C03638=1064.079,67.653,428.198,172.244,27.907,155.137
C03639=1064.085,67.903,428.181,172.246,27.909,155.137
C03640=1064.091,68.152,428.163,172.246,27.912,155.138
C03641=1064.097,68.401,428.146,172.248,27.915,155.138
C03642=1064.103,68.650,428.128,172.249,27.917,155.139
C03643=1064.109,68.899,428.111,172.251,27.920,155.139
C03644=1064.115,69.150,428.094,172.252,27.923,155.139
C03645=1064.120,69.399,428.076,172.254,27.925,155.140
C03646=1064.127,69.648,428.059,172.256,27.928,155.140
C03647=1064.133,69.897,428.041,172.257,27.931,155.141
C03648=1064.138,70.146,428.024,172.259,27.934,155.141
C03649=1064.144,70.396,428.006,172.259,27.936,155.141
C03650=1064.150,70.645,427.989,172.261,27.939,155.142
C03651=1064.157,70.894,427.971,172.262,27.941,155.142
C03652=1064.162,71.143,427.953,172.264,27.944,155.142
C03653=1064.168,71.393,427.935,172.265,27.947,155.143
C03654=1064.174,71.642,427.918,172.267,27.950,155.143
C03655=1064.180,71.891,427.901,172.269,27.952,155.144
C03656=1064.186,72.141,427.883,172.270,27.955,155.144
C03657=1064.192,72.390,427.865,172.272,27.958,155.144
C03658=1064.198,72.640,427.847,172.272,27.961,155.145
C03659=1064.203,72.889,427.830,172.274,27.963,155.145
C03660=1064.210,73.138,427.812,172.275,27.966,155.146
C03661=1064.216,73.387,427.795,172.277,27.968,155.146
C03662=1064.222,73.637,427.777,172.279,27.971,155.146
C03663=1064.227,73.886,427.759,172.280,27.974,155.147
C03664=1064.233,74.136,427.741,172.282,27.977,155.147
C03665=1064.239,74.385,427.724,172.283,27.980,155.147
C03666=1064.245,74.634,427.706,172.285,27.982,155.148
C03667=1064.251,74.883,427.689,172.285,27.984,155.148
C03668=1064.257,75.133,427.671,172.287,27.987,155.149
C03669=1064.263,75.382,427.653,172.289,27.990,155.149
C03670=1064.269,75.632,427.636,172.290,27.993,155.149
C03671=1064.275,75.881,427.618,172.292,27.996,155.150
C03672=1064.281,76.130,427.599,172.293,27.998,155.150
C03673=1064.287,76.379,427.582,172.295,28.001,155.151
C03674=1064.293,76.629,427.564,172.296,28.003,155.151
C03675=1064.299,76.877,427.547,172.298,28.006,155.151
C03676=1064.305,77.127,427.529,172.299,28.009,155.152
C03677=1064.311,77.376,427.511,172.300,28.011,155.152
C03678=1064.317,77.626,427.493,172.302,28.014,155.152
C03679=1064.323,77.874,427.475,172.303,28.017,155.153
C03680=1064.329,78.159,427.455,172.305,28.020,155.153
C03681=1064.336,78.442,427.434,172.307,28.023,155.154
C03682=1064.343,78.726,427.414,172.309,28.026,155.154
C03683=1064.349,79.010,427.394,172.310,28.029,155.155
C03684=1064.355,79.259,427.376,172.312,28.032,155.155
C03685=1064.361,79.508,427.358,172.313,28.035,155.155
C03686=1064.367,79.757,427.340,172.315,28.037,155.156
C03687=1064.373,80.007,427.322,172.315,28.040,155.156
C03688=1064.379,80.256,427.304,172.317,28.043,155.157
C03689=1064.384,80.506,427.286,172.319,28.046,155.157
C03690=1064.390,80.755,427.267,172.320,28.048,155.157
C03691=1064.396,81.004,427.249,172.322,28.051,155.158
C03692=1064.402,81.254,427.232,172.323,28.054,155.158
C03693=1064.408,81.503,427.213,172.325,28.057,155.159
C03694=1064.414,81.752,427.196,172.326,28.059,155.159
C03695=1064.420,82.001,427.178,172.328,28.062,155.159
C03696=1064.426,82.250,427.159,172.329,28.065,155.160
C03697=1064.432,82.500,427.142,172.330,28.068,155.160
C03698=1064.437,82.750,427.123,172.332,28.070,155.161
C03699=1064.443,82.998,427.105,172.333,28.073,155.161
C03700=1064.449,83.248,427.087,172.335,28.075,155.161
C03701=1064.455,83.497,427.069,172.336,28.078,155.162
C03702=1064.461,83.746,427.051,172.338,28.081,155.162
C03703=1064.467,83.996,427.033,172.339,28.084,155.162
C03704=1064.473,84.245,427.015,172.341,28.087,155.163
C03705=1064.479,84.494,426.996,172.343,28.089,155.163
C03706=1064.484,84.743,426.978,172.344,28.092,155.164
C03707=1064.490,84.992,426.960,172.346,28.095,155.164
C03708=1064.497,85.242,426.942,172.346,28.097,155.165
C03709=1064.502,85.491,426.924,172.348,28.100,155.165
C03710=1064.509,85.740,426.905,172.350,28.102,155.165
C03711=1064.515,85.990,426.888,172.351,28.105,155.166
C03712=1064.520,86.239,426.869,172.353,28.108,155.166
C03713=1064.526,86.488,426.851,172.354,28.111,155.166
C03714=1064.532,86.738,426.832,172.356,28.114,155.167
C03715=1064.538,86.987,426.814,172.357,28.116,155.167
C03716=1064.544,87.236,426.796,172.359,28.119,155.168
C03717=1064.550,87.485,426.778,172.360,28.122,155.168
C03718=1064.555,87.734,426.759,172.362,28.124,155.168
C03719=1064.562,87.984,426.741,172.364,28.127,155.169
C03720=1064.568,88.233,426.722,172.364,28.129,155.169
C03721=1064.574,88.482,426.705,172.366,28.132,155.170
C03722=1064.580,88.731,426.686,172.367,28.135,155.170
C03723=1064.585,88.981,426.668,172.369,28.138,155.170
C03724=1064.591,89.230,426.649,172.370,28.141,155.171
C03725=1064.597,89.479,426.631,172.372,28.143,155.171
C03726=1064.604,89.729,426.613,172.374,28.146,155.171
C03727=1064.610,89.978,426.594,172.375,28.148,155.172
C03728=1064.615,90.227,426.576,172.377,28.151,155.172
C03729=1064.621,90.476,426.557,172.378,28.154,155.173
C03730=1064.627,90.726,426.539,172.380,28.157,155.173
C03731=1064.633,90.974,426.521,172.382,28.159,155.173
C03732=1064.639,91.224,426.502,172.382,28.162,155.174
C03733=1064.645,91.474,426.484,172.384,28.165,155.174
C03734=1064.650,91.722,426.465,172.385,28.168,155.175
C03735=1064.657,91.971,426.446,172.387,28.170,155.175
C03736=1064.663,92.221,426.429,172.388,28.173,155.175
C03737=1064.668,92.471,426.409,172.390,28.175,155.176
C03738=1064.674,92.719,426.391,172.392,28.178,155.176
C03739=1064.680,92.969,426.372,172.393,28.181,155.177
C03740=1064.686,93.218,426.354,172.395,28.184,155.177
C03741=1064.691,93.467,426.335,172.396,28.186,155.177
C03742=1064.697,93.717,426.317,172.398,28.189,155.178
C03743=1064.704,93.966,426.298,172.399,28.192,155.178
C03744=1064.710,94.250,426.277,172.401,28.195,155.179
C03745=1064.716,94.533,426.256,172.402,28.198,155.179
C03746=1064.724,94.817,426.234,172.404,28.201,155.180
C03747=1064.730,95.101,426.213,172.406,28.204,155.180
C03748=1064.736,95.351,426.195,172.407,28.207,155.180
C03749=1064.742,95.599,426.177,172.409,28.210,155.181
C03750=1064.747,95.848,426.157,172.410,28.213,155.181
C03751=1064.754,96.098,426.139,172.412,28.215,155.182
C03752=1064.760,96.347,426.119,172.413,28.218,155.182
C03753=1064.765,96.596,426.102,172.415,28.221,155.182
C03754=1064.771,96.845,426.083,172.416,28.224,155.183
C03755=1064.777,97.095,426.064,172.418,28.226,155.183
C03756=1064.783,97.344,426.045,172.420,28.229,155.183
C03757=1064.789,97.593,426.026,172.421,28.231,155.184
C03758=1064.794,97.842,426.007,172.423,28.234,155.184
C03759=1064.801,98.092,425.989,172.424,28.237,155.185
C03760=1064.806,98.341,425.970,172.426,28.240,155.185
C03761=1064.813,98.590,425.951,172.428,28.243,155.185
C03762=1064.818,98.840,425.932,172.429,28.245,155.186
C03763=1064.824,99.088,425.914,172.430,28.248,155.186
C03764=1064.830,99.337,425.895,172.431,28.251,155.187
C03765=1064.836,99.587,425.876,172.433,28.253,155.187
C03766=1064.842,99.836,425.857,172.435,28.256,155.187
C03767=1064.848,100.085,425.838,172.436,28.258,155.188
C03768=1064.854,100.335,425.819,172.438,28.261,155.188
C03769=1064.860,100.584,425.801,172.439,28.264,155.189
C03770=1064.865,100.833,425.782,172.441,28.267,155.189
C03771=1064.872,101.082,425.763,172.442,28.269,155.189
C03772=1064.877,101.332,425.744,172.444,28.272,155.190
C03773=1064.884,101.581,425.725,172.446,28.275,155.190
C03774=1064.889,101.830,425.706,172.447,28.278,155.191
C03775=1064.895,102.079,425.687,172.449,28.281,155.191
C03776=1064.900,102.328,425.668,172.450,28.283,155.191
C03777=1064.907,102.577,425.649,172.452,28.286,155.192
C03778=1064.912,102.827,425.630,172.453,28.289,155.192
C03779=1064.918,103.076,425.611,172.455,28.292,155.193
C03780=1064.924,103.325,425.592,172.457,28.294,155.193
C03781=1064.930,103.574,425.573,172.458,28.297,155.193
C03782=1064.936,103.823,425.553,172.460,28.300,155.194
C03783=1064.941,104.072,425.534,172.460,28.302,155.194
C03784=1064.948,104.322,425.516,172.462,28.305,155.195
C03785=1064.953,104.571,425.496,172.464,28.307,155.195
C03786=1064.959,104.820,425.477,172.465,28.310,155.195
C03787=1064.965,105.070,425.458,172.467,28.313,155.196
C03788=1064.971,105.318,425.440,172.468,28.316,155.196
C03789=1064.976,105.568,425.420,172.470,28.318,155.197
C03790=1064.982,105.817,425.401,172.471,28.321,155.197
C03791=1064.988,106.066,425.381,172.473,28.324,155.197
C03792=1064.994,106.315,425.362,172.475,28.327,155.198
C03793=1065.000,106.564,425.343,172.476,28.330,155.198
C03794=1065.006,106.814,425.324,172.478,28.332,155.199
C03795=1065.011,107.063,425.305,172.479,28.335,155.199
C03796=1065.018,107.312,425.286,172.481,28.338,155.199
C03797=1065.024,107.561,425.266,172.483,28.341,155.200
C03798=1065.030,107.811,425.247,172.484,28.343,155.200
C03799=1065.035,108.059,425.228,172.486,28.346,155.201
C03800=1065.041,108.309,425.209,172.487,28.349,155.201
C03801=1065.047,108.558,425.190,172.489,28.352,155.201
C03802=1065.053,108.807,425.170,172.491,28.354,155.202
C03803=1065.058,109.056,425.151,172.492,28.357,155.202
C03804=1065.064,109.306,425.132,172.494,28.359,155.202
C03805=1065.071,109.555,425.113,172.495,28.362,155.203
C03806=1065.077,109.804,425.093,172.497,28.365,155.203
C03807=1065.082,110.053,425.074,172.498,28.368,155.204
C03808=1065.089,110.337,425.052,172.500,28.370,155.204
C03809=1065.096,110.621,425.030,172.502,28.374,155.205
C03810=1065.102,110.904,425.008,172.503,28.377,155.205
C03811=1065.109,111.189,424.985,172.506,28.380,155.205
C03812=1065.115,111.438,424.966,172.507,28.383,155.206
C03813=1065.121,111.688,424.947,172.509,28.386,155.206
C03814=1065.128,111.936,424.928,172.510,28.388,155.207
C03815=1065.133,112.185,424.908,172.512,28.391,155.207
C03816=1065.138,112.434,424.889,172.513,28.394,155.207
C03817=1065.144,112.683,424.870,172.515,28.397,155.208
C03818=1065.150,112.932,424.850,172.517,28.399,155.208
C03819=1065.156,113.181,424.830,172.518,28.402,155.209
C03820=1065.162,113.431,424.811,172.520,28.404,155.209
C03821=1065.167,113.680,424.792,172.521,28.407,155.209
C03822=1065.173,113.929,424.772,172.523,28.410,155.210
C03823=1065.179,114.178,424.753,172.525,28.413,155.210
C03824=1065.185,114.427,424.733,172.526,28.415,155.211
C03825=1065.191,114.677,424.713,172.528,28.418,155.211
C03826=1065.197,114.925,424.693,172.529,28.421,155.211
C03827=1065.202,115.175,424.674,172.531,28.424,155.212
C03828=1065.208,115.424,424.654,172.533,28.426,155.212
C03829=1065.213,115.673,424.634,172.534,28.430,155.213
C03830=1065.219,115.923,424.615,172.536,28.433,155.213
C03831=1065.225,116.172,424.595,172.537,28.435,155.214
C03832=1065.231,116.420,424.575,172.539,28.438,155.214
C03833=1065.237,116.670,424.556,172.540,28.441,155.214
C03834=1065.242,116.919,424.535,172.542,28.444,155.215
C03835=1065.248,117.168,424.516,172.544,28.446,155.215
C03836=1065.254,117.417,424.496,172.545,28.449,155.216
C03837=1065.259,117.667,424.477,172.547,28.452,155.216
C03838=1065.265,117.916,424.457,172.548,28.455,155.216
C03839=1065.271,118.165,424.438,172.550,28.457,155.217
C03840=1065.276,118.414,424.417,172.552,28.460,155.217
C03841=1065.282,118.663,424.397,172.553,28.463,155.218
C03842=1065.288,118.912,424.378,172.555,28.466,155.218
C03843=1065.294,119.161,424.358,172.556,28.468,155.218
C03844=1065.300,119.411,424.339,172.558,28.471,155.219
C03845=1065.306,119.660,424.318,172.560,28.474,155.219
C03846=1065.312,119.909,424.298,172.561,28.477,155.220
C03847=1065.317,120.159,424.279,172.563,28.479,155.220
C03848=1065.323,120.407,424.259,172.564,28.482,155.220
C03849=1065.329,120.656,424.239,172.566,28.485,155.221
C03850=1065.334,120.906,424.219,172.568,28.488,155.221
C03851=1065.340,121.155,424.199,172.569,28.490,155.222
C03852=1065.346,121.404,424.179,172.571,28.493,155.222
C03853=1065.352,121.653,424.160,172.572,28.496,155.222
C03854=1065.358,121.902,424.140,172.574,28.499,155.223
C03855=1065.363,122.151,424.119,172.575,28.501,155.223
C03856=1065.369,122.401,424.100,172.577,28.504,155.224
C03857=1065.375,122.650,424.080,172.579,28.507,155.224
C03858=1065.381,122.899,424.060,172.580,28.510,155.224
C03859=1065.387,123.148,424.039,172.582,28.512,155.225
C03860=1065.392,123.397,424.020,172.583,28.515,155.225
C03861=1065.398,123.646,424.000,172.585,28.518,155.226
C03862=1065.404,123.895,423.980,172.587,28.521,155.226
C03863=1065.410,124.144,423.960,172.588,28.523,155.226
C03864=1065.416,124.394,423.940,172.590,28.526,155.227
C03865=1065.422,124.643,423.920,172.591,28.529,155.227
C03866=1065.428,124.892,423.900,172.593,28.532,155.228
C03867=1065.434,125.141,423.880,172.595,28.534,155.228
C03868=1065.439,125.390,423.859,172.596,28.537,155.228
C03869=1065.445,125.639,423.840,172.598,28.539,155.229
C03870=1065.451,125.889,423.820,172.600,28.542,155.229
C03871=1065.457,126.138,423.800,172.601,28.545,155.230
C03872=1065.463,126.421,423.776,172.604,28.548,155.230
C03873=1065.470,126.705,423.754,172.605,28.551,155.230
C03874=1065.477,126.989,423.731,172.607,28.554,155.231
C03875=1065.484,127.272,423.708,172.609,28.557,155.231
C03876=1065.489,127.521,423.688,172.611,28.560,155.232
C03877=1065.496,127.771,423.667,172.612,28.563,155.232
C03878=1065.502,128.019,423.647,172.614,28.566,155.233
C03879=1065.507,128.269,423.628,172.616,28.568,155.233
C03880=1065.513,128.518,423.608,172.617,28.571,155.233
C03881=1065.519,128.767,423.587,172.619,28.574,155.234
C03882=1065.525,129.016,423.567,172.620,28.577,155.234
C03883=1065.531,129.265,423.547,172.622,28.579,155.235
C03884=1065.537,129.514,423.527,172.624,28.582,155.235
C03885=1065.543,129.764,423.507,172.625,28.584,155.235
C03886=1065.548,130.013,423.486,172.627,28.587,155.236
C03887=1065.554,130.262,423.466,172.629,28.590,155.236
C03888=1065.560,130.510,423.446,172.630,28.593,155.237
C03889=1065.566,130.760,423.425,172.632,28.595,155.237
C03890=1065.572,131.009,423.405,172.634,28.598,155.237
C03891=1065.578,131.258,423.385,172.636,28.601,155.238
C03892=1065.584,131.508,423.364,172.638,28.604,155.238
C03893=1065.590,131.757,423.344,172.639,28.607,155.239
C03894=1065.596,132.005,423.324,172.641,28.609,155.239
C03895=1065.601,132.254,423.304,172.642,28.612,155.239
C03896=1065.608,132.504,423.283,172.644,28.615,155.240
C03897=1065.614,132.753,423.262,172.646,28.617,155.240
C03898=1065.619,133.002,423.242,172.647,28.620,155.241
C03899=1065.625,133.250,423.222,172.649,28.623,155.241
C03900=1065.631,133.500,423.201,172.650,28.626,155.241
C03901=1065.637,133.749,423.181,172.652,28.628,155.242
C03902=1065.642,133.998,423.160,172.654,28.631,155.242
C03903=1065.648,134.247,423.140,172.656,28.634,155.243
C03904=1065.654,134.496,423.119,172.658,28.637,155.243
C03905=1065.659,134.745,423.098,172.659,28.640,155.243
C03906=1065.665,134.994,423.078,172.661,28.642,155.244
C03907=1065.671,135.244,423.057,172.663,28.645,155.244
C03908=1065.677,135.493,423.037,172.664,28.648,155.245
C03909=1065.682,135.742,423.017,172.666,28.651,155.245
C03910=1065.689,135.991,422.996,172.667,28.653,155.245
C03911=1065.695,136.240,422.975,172.669,28.656,155.246
C03912=1065.700,136.489,422.955,172.671,28.659,155.246
C03913=1065.706,136.739,422.934,172.672,28.662,155.247
C03914=1065.712,136.987,422.913,172.675,28.665,155.247
C03915=1065.718,137.236,422.893,172.676,28.667,155.247
C03916=1065.724,137.486,422.872,172.678,28.670,155.248
C03917=1065.729,137.735,422.852,172.680,28.673,155.248
C03918=1065.735,137.983,422.831,172.681,28.675,155.249
C03919=1065.741,138.233,422.810,172.683,28.678,155.249
C03920=1065.747,138.482,422.789,172.684,28.681,155.249
C03921=1065.753,138.730,422.769,172.686,28.684,155.250
C03922=1065.759,138.980,422.748,172.688,28.686,155.250
C03923=1065.764,139.229,422.727,172.689,28.689,155.251
C03924=1065.770,139.477,422.707,172.692,28.692,155.251
C03925=1065.776,139.727,422.686,172.693,28.695,155.251
C03926=1065.781,139.976,422.665,172.695,28.698,155.252
C03927=1065.788,140.224,422.644,172.697,28.700,155.252
C03928=1065.793,140.474,422.624,172.698,28.703,155.253
C03929=1065.799,140.723,422.603,172.700,28.706,155.253
C03930=1065.805,140.973,422.581,172.702,28.709,155.253
C03931=1065.810,141.222,422.561,172.703,28.711,155.254
C03932=1065.816,141.470,422.540,172.705,28.714,155.254
C03933=1065.822,141.720,422.519,172.707,28.717,155.255
C03934=1065.828,141.968,422.498,172.709,28.720,155.255
C03935=1065.833,142.217,422.477,172.711,28.722,155.255
C03936=1065.840,142.501,422.453,172.712,28.726,155.256
C03937=1065.846,142.785,422.430,172.715,28.729,155.256
C03938=1065.853,143.069,422.406,172.716,28.732,155.257
C03939=1065.860,143.351,422.382,172.718,28.735,155.257
C03940=1065.866,143.601,422.361,172.720,28.738,155.258
C03941=1065.871,143.850,422.340,172.722,28.741,155.258
C03942=1065.877,144.099,422.319,172.724,28.744,155.259
C03943=1065.883,144.348,422.298,172.725,28.746,155.259
C03944=1065.889,144.598,422.277,172.727,28.749,155.259
C03945=1065.894,144.846,422.255,172.728,28.752,155.260
C03946=1065.900,145.095,422.235,172.730,28.755,155.260
C03947=1065.906,145.344,422.214,172.733,28.758,155.261
C03948=1065.912,145.593,422.193,172.734,28.760,155.261
C03949=1065.918,145.843,422.172,172.736,28.763,155.261
C03950=1065.923,146.091,422.150,172.737,28.766,155.262
C03951=1065.929,146.341,422.129,172.739,28.769,155.262
C03952=1065.935,146.589,422.108,172.741,28.771,155.263
C03953=1065.941,146.839,422.088,172.742,28.774,155.263
C03954=1065.947,147.087,422.067,172.745,28.777,155.263
C03955=1065.953,147.337,422.045,172.746,28.780,155.264
C03956=1065.958,147.586,422.024,172.748,28.782,155.264
C03957=1065.964,147.835,422.003,172.750,28.785,155.265
C03958=1065.970,148.083,421.981,172.751,28.788,155.265
C03959=1065.976,148.333,421.961,172.753,28.791,155.265
C03960=1065.981,148.582,421.939,172.756,28.794,155.266
C03961=1065.988,148.831,421.918,172.757,28.796,155.266
C03962=1065.993,149.080,421.897,172.759,28.799,155.267
C03963=1065.999,149.329,421.875,172.760,28.802,155.267
C03964=1066.005,149.578,421.854,172.762,28.804,155.267
C03965=1066.011,149.827,421.833,172.764,28.807,155.268
C03966=1066.016,150.076,421.812,172.766,28.810,155.268
C03967=1066.022,150.325,421.790,172.768,28.813,155.269
C03968=1066.028,150.574,421.769,172.769,28.816,155.269
C03969=1066.034,150.823,421.747,172.771,28.819,155.270
C03970=1066.039,151.072,421.726,172.773,28.822,155.270
C03971=1066.045,151.321,421.705,172.774,28.824,155.270
C03972=1066.050,151.570,421.683,172.777,28.827,155.271
C03973=1066.056,151.819,421.662,172.778,28.830,155.271
C03974=1066.062,152.068,421.640,172.780,28.833,155.272
C03975=1066.068,152.317,421.619,172.782,28.835,155.272
C03976=1066.074,152.566,421.598,172.783,28.838,155.272
C03977=1066.079,152.815,421.577,172.786,28.841,155.273
C03978=1066.085,153.064,421.555,172.788,28.844,155.273
C03979=1066.091,153.313,421.534,172.789,28.847,155.274
C03980=1066.097,153.562,421.512,172.791,28.850,155.274
C03981=1066.102,153.811,421.490,172.792,28.853,155.275
C03982=1066.108,154.060,421.469,172.794,28.855,155.275
C03983=1066.114,154.309,421.447,172.797,28.858,155.275
C03984=1066.120,154.558,421.426,172.798,28.861,155.276
C03985=1066.126,154.807,421.404,172.800,28.864,155.276
C03986=1066.132,155.056,421.383,172.801,28.866,155.277
C03987=1066.138,155.306,421.362,172.803,28.869,155.277
C03988=1066.142,155.554,421.340,172.806,28.872,155.277
C03989=1066.149,155.804,421.318,172.807,28.875,155.278
C03990=1066.154,156.052,421.297,172.809,28.878,155.278
C03991=1066.160,156.301,421.275,172.811,28.880,155.279
C03992=1066.166,156.551,421.253,172.813,28.884,155.279
C03993=1066.171,156.799,421.232,172.815,28.887,155.280
C03994=1066.177,157.049,421.210,172.816,28.889,155.280
C03995=1066.183,157.297,421.189,172.818,28.892,155.280
C03996=1066.189,157.546,421.166,172.820,28.895,155.281
C03997=1066.195,157.795,421.145,172.822,28.898,155.281
C03998=1066.200,158.044,421.123,172.824,28.900,155.282
C03999=1066.206,158.293,421.101,172.825,28.903,155.282
C04000=1066.213,158.577,421.076,172.828,28.907,155.282
C04001=1066.219,158.859,421.052,172.830,28.910,155.283
C04002=1066.226,159.143,421.027,172.832,28.913,155.283
C04003=1066.233,159.427,421.002,172.834,28.916,155.284
C04004=1066.238,159.675,420.981,172.835,28.919,155.284
C04005=1066.244,159.924,420.959,172.838,28.922,155.285
C04006=1066.250,160.174,420.937,172.840,28.924,155.285
C04007=1066.255,160.422,420.916,172.841,28.927,155.286
C04008=1066.261,160.671,420.894,172.843,28.930,155.286
C04009=1066.267,160.921,420.872,172.845,28.933,155.286
C04010=1066.273,161.169,420.850,172.847,28.936,155.287
C04011=1066.279,161.418,420.828,172.849,28.939,155.287
C04012=1066.284,161.668,420.806,172.850,28.942,155.288
C04013=1066.289,161.916,420.784,172.853,28.944,155.288
C04014=1066.296,162.165,420.762,172.854,28.948,155.289
C04015=1066.300,162.414,420.740,172.856,28.950,155.289
C04016=1066.307,162.663,420.718,172.858,28.953,155.289
C04017=1066.312,162.913,420.696,172.859,28.956,155.290
C04018=1066.317,163.161,420.673,172.862,28.959,155.290
C04019=1066.323,163.410,420.652,172.863,28.962,155.291
C04020=1066.329,163.659,420.629,172.865,28.965,155.291
C04021=1066.334,163.908,420.607,172.867,28.968,155.292
C04022=1066.340,164.157,420.585,172.869,28.971,155.292
C04023=1066.345,164.406,420.563,172.871,28.974,155.292
C04024=1066.351,164.655,420.540,172.873,28.976,155.293
C04025=1066.357,164.904,420.519,172.874,28.980,155.293
C04026=1066.362,165.153,420.497,172.877,28.983,155.294
C04027=1066.368,165.401,420.475,172.878,28.985,155.294
C04028=1066.374,165.651,420.452,172.880,28.988,155.295
C04029=1066.379,165.900,420.430,172.883,28.992,155.295
C04030=1066.385,166.148,420.408,172.884,28.994,155.295
C04031=1066.390,166.398,420.386,172.886,28.997,155.296
C04032=1066.396,166.647,420.363,172.887,29.000,155.296
C04033=1066.402,166.895,420.342,172.890,29.003,155.297
C04034=1066.407,167.144,420.319,172.892,29.006,155.297
C04035=1066.413,167.393,420.296,172.893,29.009,155.298
C04036=1066.419,167.642,420.274,172.895,29.011,155.298
C04037=1066.424,167.891,420.252,172.897,29.015,155.299
C04038=1066.429,168.140,420.230,172.899,29.018,155.299
C04039=1066.435,168.389,420.207,172.901,29.020,155.299
C04040=1066.441,168.638,420.185,172.903,29.023,155.300
C04041=1066.446,168.887,420.163,172.905,29.026,155.300
C04042=1066.452,169.136,420.140,172.907,29.029,155.301
C04043=1066.458,169.385,420.118,172.908,29.032,155.301
C04044=1066.464,169.634,420.095,172.911,29.035,155.301
C04045=1066.469,169.882,420.073,172.912,29.038,155.302
C04046=1066.475,170.131,420.051,172.914,29.041,155.302
C04047=1066.481,170.381,420.029,172.917,29.044,155.303
C04048=1066.487,170.629,420.006,172.918,29.046,155.303
C04049=1066.492,170.879,419.984,172.920,29.049,155.304
C04050=1066.498,171.127,419.962,172.922,29.053,155.304
C04051=1066.504,171.376,419.939,172.924,29.055,155.305
C04052=1066.509,171.625,419.917,172.926,29.058,155.305
C04053=1066.515,171.874,419.894,172.927,29.061,155.305
C04054=1066.521,172.123,419.871,172.930,29.064,155.306
C04055=1066.527,172.372,419.849,172.932,29.067,155.306
C04056=1066.532,172.620,419.826,172.933,29.070,155.307
C04057=1066.538,172.869,419.804,172.936,29.073,155.307
C04058=1066.544,173.119,419.782,172.937,29.075,155.307
C04059=1066.549,173.367,419.759,172.939,29.079,155.308
C04060=1066.555,173.616,419.736,172.942,29.081,155.308
C04061=1066.561,173.866,419.714,172.943,29.084,155.309
C04062=1066.567,174.114,419.691,172.945,29.087,155.309
C04063=1066.573,174.363,419.668,172.947,29.090,155.310
C04064=1066.579,174.646,419.643,172.949,29.093,155.310
C04065=1066.586,174.929,419.618,172.952,29.097,155.311
C04066=1066.592,175.212,419.592,172.954,29.100,155.311
C04067=1066.598,175.495,419.566,172.956,29.103,155.312
C04068=1066.604,175.744,419.543,172.958,29.106,155.312
C04069=1066.610,175.992,419.521,172.960,29.109,155.312
C04070=1066.616,176.241,419.498,172.962,29.112,155.313
C04071=1066.622,176.491,419.476,172.964,29.115,155.313
C04072=1066.627,176.739,419.453,172.966,29.118,155.314
C04073=1066.633,176.988,419.430,172.968,29.121,155.314
C04074=1066.640,177.237,419.408,172.970,29.123,155.315
C04075=1066.645,177.486,419.385,172.972,29.126,155.315
C04076=1066.651,177.735,419.362,172.974,29.130,155.316
C04077=1066.657,177.984,419.339,172.976,29.132,155.316
C04078=1066.662,178.233,419.317,172.978,29.135,155.316
C04079=1066.669,178.482,419.294,172.980,29.138,155.317
C04080=1066.674,178.731,419.271,172.982,29.141,155.317
C04081=1066.680,178.980,419.248,172.983,29.144,155.318
C04082=1066.686,179.228,419.225,172.986,29.147,155.318
C04083=1066.692,179.477,419.202,172.988,29.149,155.318
C04084=1066.697,179.726,419.180,172.990,29.152,155.319
C04085=1066.704,179.975,419.157,172.992,29.155,155.319
C04086=1066.710,180.224,419.134,172.994,29.158,155.320
C04087=1066.715,180.473,419.111,172.996,29.161,155.320
C04088=1066.721,180.722,419.088,172.998,29.164,155.321
C04089=1066.727,180.970,419.065,173.000,29.167,155.321
C04090=1066.732,181.219,419.042,173.002,29.170,155.321
C04091=1066.739,181.468,419.020,173.004,29.173,155.322
C04092=1066.745,181.717,418.997,173.006,29.176,155.322
C04093=1066.750,181.966,418.974,173.008,29.178,155.323
C04094=1066.756,182.215,418.951,173.011,29.181,155.323
C04095=1066.762,182.464,418.928,173.012,29.184,155.324
C04096=1066.768,182.713,418.905,173.014,29.187,155.324
C04097=1066.775,182.962,418.883,173.016,29.190,155.324
C04098=1066.780,183.211,418.860,173.018,29.193,155.325
C04099=1066.786,183.459,418.837,173.021,29.196,155.325
C04100=1066.792,183.708,418.814,173.022,29.198,155.326
C04101=1066.798,183.957,418.790,173.025,29.201,155.326
C04102=1066.804,184.206,418.767,173.027,29.205,155.327
C04103=1066.809,184.454,418.744,173.028,29.207,155.327
C04104=1066.816,184.704,418.721,173.031,29.210,155.327
C04105=1066.821,184.953,418.698,173.032,29.213,155.328
C04106=1066.827,185.202,418.675,173.035,29.216,155.328
C04107=1066.832,185.450,418.651,173.037,29.219,155.329
C04108=1066.838,185.699,418.628,173.038,29.222,155.329
C04109=1066.844,185.948,418.605,173.041,29.225,155.330
C04110=1066.849,186.197,418.581,173.043,29.228,155.330
C04111=1066.855,186.446,418.558,173.045,29.231,155.331
C04112=1066.861,186.695,418.535,173.047,29.235,155.331
C04113=1066.866,186.944,418.511,173.049,29.238,155.331
C04114=1066.871,187.193,418.488,173.051,29.241,155.332
C04115=1066.877,187.441,418.465,173.053,29.243,155.332
C04116=1066.883,187.690,418.442,173.055,29.247,155.333
C04117=1066.888,187.939,418.418,173.057,29.250,155.333
C04118=1066.894,188.187,418.394,173.059,29.253,155.334
C04119=1066.899,188.437,418.371,173.061,29.256,155.334
C04120=1066.905,188.685,418.348,173.064,29.259,155.335
C04121=1066.911,188.934,418.324,173.065,29.262,155.335
C04122=1066.916,189.183,418.301,173.068,29.265,155.336
C04123=1066.922,189.431,418.277,173.070,29.268,155.336
C04124=1066.928,189.681,418.254,173.071,29.271,155.337
C04125=1066.933,189.930,418.230,173.074,29.274,155.337
C04126=1066.939,190.178,418.207,173.075,29.277,155.337
C04127=1066.945,190.427,418.184,173.078,29.280,155.338
C04128=1066.951,190.710,418.156,173.081,29.284,155.338
C04129=1066.958,190.992,418.130,173.082,29.287,155.339
C04130=1066.964,191.274,418.103,173.085,29.291,155.340
C04131=1066.971,191.557,418.076,173.087,29.294,155.340
C04132=1066.976,191.806,418.053,173.089,29.297,155.341
C04133=1066.982,192.055,418.029,173.092,29.300,155.341
C04134=1066.987,192.303,418.006,173.093,29.303,155.341
C04135=1066.994,192.552,417.982,173.096,29.306,155.342
C04136=1066.999,192.802,417.958,173.097,29.310,155.342
C04137=1067.005,193.050,417.934,173.100,29.312,155.343
C04138=1067.011,193.299,417.912,173.102,29.315,155.343
C04139=1067.016,193.547,417.887,173.104,29.319,155.344
C04140=1067.022,193.797,417.864,173.106,29.321,155.344
C04141=1067.028,194.046,417.840,173.108,29.325,155.345
C04142=1067.034,194.294,417.816,173.110,29.327,155.345
C04143=1067.039,194.543,417.792,173.113,29.331,155.346
C04144=1067.045,194.791,417.769,173.114,29.334,155.346
C04145=1067.051,195.041,417.746,173.117,29.337,155.346
C04146=1067.056,195.290,417.721,173.119,29.340,155.347
C04147=1067.062,195.538,417.698,173.121,29.343,155.347
C04148=1067.067,195.787,417.674,173.123,29.346,155.348
C04149=1067.074,196.036,417.650,173.125,29.349,155.348
C04150=1067.079,196.285,417.626,173.127,29.352,155.349
C04151=1067.085,196.533,417.602,173.130,29.355,155.349
C04152=1067.092,196.782,417.579,173.131,29.358,155.350
C04153=1067.097,197.031,417.555,173.134,29.362,155.350
C04154=1067.103,197.279,417.531,173.136,29.364,155.351
C04155=1067.108,197.529,417.507,173.138,29.368,155.351
C04156=1067.115,197.778,417.483,173.141,29.371,155.352
C04157=1067.120,198.026,417.459,173.142,29.373,155.352
C04158=1067.126,198.274,417.435,173.145,29.377,155.352
C04159=1067.132,198.524,417.411,173.147,29.379,155.353
C04160=1067.138,198.773,417.388,173.149,29.383,155.353
C04161=1067.143,199.021,417.364,173.151,29.386,155.354
C04162=1067.150,199.270,417.340,173.154,29.389,155.354
C04163=1067.155,199.519,417.315,173.155,29.392,155.355
C04164=1067.161,199.767,417.292,173.158,29.395,155.355
C04165=1067.166,200.017,417.268,173.160,29.398,155.356
C04166=1067.173,200.265,417.244,173.162,29.401,155.356
C04167=1067.178,200.514,417.219,173.165,29.404,155.357
C04168=1067.184,200.763,417.196,173.166,29.407,155.357
C04169=1067.190,201.011,417.172,173.169,29.410,155.357
C04170=1067.196,201.260,417.147,173.171,29.413,155.358
C04171=1067.202,201.509,417.123,173.173,29.416,155.358
C04172=1067.208,201.758,417.099,173.175,29.420,155.359
C04173=1067.214,202.006,417.075,173.177,29.422,155.359
C04174=1067.220,202.255,417.051,173.180,29.426,155.360
C04175=1067.226,202.504,417.027,173.182,29.429,155.360
C04176=1067.231,202.753,417.002,173.184,29.432,155.361
C04177=1067.237,203.001,416.979,173.186,29.435,155.361
C04178=1067.243,203.250,416.954,173.189,29.438,155.362
C04179=1067.248,203.499,416.930,173.190,29.441,155.362
C04180=1067.253,203.747,416.906,173.193,29.445,155.363
C04181=1067.259,203.997,416.881,173.195,29.448,155.363
C04182=1067.265,204.245,416.857,173.197,29.451,155.364
C04183=1067.271,204.494,416.833,173.200,29.454,155.364
C04184=1067.277,204.743,416.808,173.201,29.457,155.365
C04185=1067.282,204.991,416.784,173.204,29.460,155.365
C04186=1067.288,205.240,416.760,173.206,29.464,155.366
C04187=1067.294,205.489,416.736,173.208,29.467,155.366
C04188=1067.300,205.738,416.711,173.211,29.470,155.367
C04189=1067.305,205.987,416.687,173.212,29.473,155.367
C04190=1067.311,206.235,416.662,173.215,29.477,155.368
C04191=1067.317,206.484,416.638,173.218,29.480,155.368
C04192=1067.341,207.529,416.535,173.367,29.555,155.372
C04193=1067.347,207.746,416.513,173.369,29.559,155.373
C04194=1067.352,207.964,416.491,173.370,29.562,155.373
C04195=1067.357,208.181,416.469,173.372,29.566,155.374
C04196=1067.362,208.398,416.447,173.374,29.569,155.375
C04197=1067.367,208.615,416.425,173.375,29.573,155.375
C04198=1067.372,208.833,416.403,173.377,29.576,155.376
C04199=1067.377,209.050,416.381,173.379,29.580,155.376
C04200=1067.382,209.268,416.359,173.381,29.583,155.377
C04201=1067.389,209.516,416.333,173.383,29.587,155.378
C04202=1067.394,209.764,416.308,173.385,29.592,155.379
C04203=1067.400,210.013,416.283,173.387,29.596,155.379
C04204=1067.407,210.262,416.258,173.389,29.600,155.380
C04205=1067.413,210.511,416.233,173.391,29.604,155.381
C04206=1067.418,210.760,416.207,173.392,29.608,155.381
C04207=1067.424,211.009,416.182,173.395,29.612,155.382
C04208=1067.430,211.257,416.157,173.396,29.616,155.383
C04209=1067.436,211.505,416.131,173.399,29.620,155.383
C04210=1067.442,211.754,416.106,173.400,29.624,155.384
C04211=1067.448,212.003,416.080,173.403,29.628,155.385
C04212=1067.454,212.252,416.055,173.405,29.632,155.385
C04213=1067.460,212.500,416.030,173.407,29.636,155.386
C04214=1067.466,212.749,416.004,173.409,29.640,155.387
C04215=1067.471,212.997,415.979,173.411,29.644,155.387
C04216=1067.477,213.246,415.953,173.413,29.648,155.388
C04217=1067.484,213.495,415.928,173.415,29.652,155.389
C04218=1067.489,213.744,415.902,173.417,29.657,155.390
C04219=1067.496,213.992,415.876,173.419,29.661,155.390
C04220=1067.501,214.241,415.850,173.421,29.665,155.391
C04221=1067.507,214.489,415.825,173.423,29.669,155.392
C04222=1067.513,214.737,415.800,173.425,29.673,155.392
C04223=1067.518,214.986,415.774,173.427,29.677,155.393
C04224=1067.525,215.235,415.748,173.429,29.681,155.394
C04225=1067.530,215.484,415.723,173.431,29.685,155.395
C04226=1067.537,215.732,415.696,173.433,29.689,155.395
C04227=1067.543,215.981,415.671,173.435,29.693,155.396
C04228=1067.548,216.230,415.645,173.437,29.697,155.397
C04229=1067.554,216.478,415.620,173.439,29.701,155.397
C04230=1067.560,216.727,415.594,173.441,29.705,155.398
C04231=1067.566,216.975,415.568,173.443,29.709,155.399
C04232=1067.573,217.224,415.543,173.446,29.714,155.399
C04233=1067.578,217.473,415.517,173.447,29.717,155.400
C04234=1067.584,217.721,415.492,173.450,29.721,155.401
C04235=1067.589,217.969,415.465,173.451,29.726,155.401
C04236=1067.596,218.218,415.440,173.454,29.730,155.402
C04237=1067.601,218.467,415.414,173.455,29.733,155.403
C04238=1067.608,218.715,415.388,173.458,29.738,155.404
C04239=1067.613,218.964,415.362,173.459,29.742,155.404
C04240=1067.619,219.213,415.336,173.462,29.746,155.405
C04241=1067.625,219.461,415.310,173.465,29.749,155.405
C04242=1067.631,219.710,415.284,173.466,29.754,155.406
C04243=1067.637,219.958,415.259,173.469,29.758,155.407
C04244=1067.643,220.207,415.232,173.470,29.762,155.408
C04245=1067.649,220.455,415.207,173.473,29.766,155.408
C04246=1067.656,220.705,415.181,173.474,29.770,155.409
C04247=1067.662,220.953,415.155,173.477,29.774,155.410
C04248=1067.667,221.202,415.129,173.479,29.777,155.410
C04249=1067.673,221.421,415.105,173.480,29.781,155.411
C04250=1067.678,221.640,415.083,173.483,29.785,155.411
C04251=1067.683,221.860,415.060,173.484,29.788,155.412
C04252=1067.688,222.080,415.037,173.486,29.792,155.413
C04253=1067.693,222.299,415.013,173.488,29.795,155.413
C04254=1067.699,222.519,414.991,173.490,29.799,155.414
C04255=1067.704,222.739,414.968,173.492,29.802,155.415
C04256=1067.709,222.959,414.944,173.494,29.806,155.415
C04257=1067.715,223.207,414.918,173.496,29.810,155.416
C04258=1067.721,223.456,414.892,173.498,29.814,155.417
C04259=1067.726,223.705,414.866,173.500,29.818,155.417
C04260=1067.733,223.953,414.840,173.502,29.822,155.418
C04261=1067.738,224.202,414.814,173.504,29.827,155.419
C04262=1067.744,224.450,414.787,173.506,29.830,155.419
C04263=1067.751,224.698,414.761,173.509,29.834,155.420
C04264=1067.756,224.947,414.735,173.511,29.839,155.421
C04265=1067.762,225.195,414.709,173.513,29.843,155.421
C04266=1067.768,225.444,414.682,173.515,29.846,155.422
C04267=1067.774,225.692,414.657,173.517,29.850,155.423
C04268=1067.780,225.941,414.630,173.519,29.855,155.424
C04269=1067.786,226.190,414.603,173.521,29.858,155.424
C04270=1067.792,226.439,414.577,173.524,29.862,155.425
C04271=1067.798,226.687,414.551,173.526,29.866,155.425
C04272=1067.804,226.935,414.524,173.528,29.871,155.426
C04273=1067.809,227.184,414.498,173.530,29.875,155.427
C04274=1067.815,227.433,414.472,173.532,29.878,155.428
C04275=1067.822,227.681,414.445,173.534,29.882,155.428
C04276=1067.828,227.930,414.419,173.536,29.887,155.429
C04277=1067.833,228.179,414.393,173.539,29.891,155.430
C04278=1067.839,228.427,414.366,173.541,29.894,155.430
C04279=1067.846,228.675,414.340,173.543,29.898,155.431
C04280=1067.852,228.923,414.313,173.545,29.903,155.432
C04281=1067.858,229.172,414.286,173.547,29.906,155.432
C04282=1067.863,229.421,414.260,173.550,29.910,155.433
C04283=1067.869,229.670,414.234,173.552,29.914,155.434
C04284=1067.876,229.918,414.208,173.554,29.918,155.434
C04285=1067.882,230.167,414.181,173.556,29.922,155.435
C04286=1067.888,230.415,414.154,173.558,29.926,155.436
C04287=1067.894,230.664,414.127,173.560,29.930,155.436
C04288=1067.899,230.912,414.101,173.563,29.935,155.437
C04289=1067.905,231.160,414.074,173.565,29.938,155.438
C04290=1067.912,231.409,414.047,173.567,29.942,155.438
C04291=1067.917,231.658,414.020,173.569,29.946,155.439
C04292=1067.923,231.906,413.994,173.571,29.951,155.440
C04293=1067.929,232.154,413.967,173.574,29.954,155.441
C04294=1067.935,232.403,413.940,173.576,29.958,155.441
C04295=1067.941,232.652,413.913,173.578,29.962,155.442
C04296=1067.947,232.900,413.887,173.580,29.966,155.443
C04297=1067.953,233.149,413.860,173.582,29.970,155.443
C04298=1067.958,233.397,413.833,173.585,29.974,155.444
C04299=1067.965,233.646,413.806,173.587,29.978,155.445
C04300=1067.970,233.894,413.780,173.589,29.982,155.445
C04301=1067.976,234.143,413.753,173.592,29.986,155.446
C04302=1067.981,234.391,413.726,173.593,29.990,155.447
C04303=1067.988,234.640,413.699,173.596,29.995,155.447
C04304=1067.993,234.889,413.672,173.598,29.998,155.448
C04305=1067.999,235.104,413.649,173.600,30.002,155.449
C04306=1068.004,235.320,413.626,173.602,30.005,155.449
C04307=1068.009,235.535,413.603,173.604,30.009,155.450
C04308=1068.014,235.751,413.579,173.606,30.013,155.450
C04309=1068.019,235.966,413.555,173.608,30.016,155.451
C04310=1068.024,236.181,413.532,173.609,30.019,155.452
C04311=1068.029,236.397,413.508,173.612,30.023,155.452
C04312=1068.035,236.613,413.485,173.614,30.026,155.453
C04313=1068.041,236.861,413.458,173.615,30.030,155.454
C04314=1068.046,237.110,413.431,173.618,30.034,155.454
C04315=1068.052,237.358,413.404,173.621,30.038,155.455
C04316=1068.058,237.607,413.377,173.622,30.042,155.456
C04317=1068.064,237.855,413.350,173.625,30.046,155.456
C04318=1068.071,238.104,413.323,173.627,30.050,155.457
C04319=1068.077,238.352,413.296,173.629,30.054,155.458
C04320=1068.082,238.600,413.269,173.632,30.058,155.458
C04321=1068.088,238.850,413.241,173.634,30.062,155.459
C04322=1068.094,239.098,413.214,173.636,30.066,155.460
C04323=1068.100,239.346,413.187,173.638,30.070,155.460
C04324=1068.106,239.595,413.160,173.641,30.074,155.461
C04325=1068.112,239.843,413.133,173.643,30.078,155.462
C04326=1068.118,240.092,413.105,173.645,30.081,155.462
C04327=1068.124,240.340,413.078,173.648,30.086,155.463
C04328=1068.130,240.588,413.051,173.649,30.090,155.464
C04329=1068.136,240.837,413.024,173.652,30.094,155.464
C04330=1068.142,241.085,412.996,173.655,30.097,155.465
C04331=1068.148,241.334,412.969,173.657,30.101,155.466
C04332=1068.154,241.582,412.942,173.659,30.106,155.466
C04333=1068.160,241.831,412.915,173.661,30.110,155.467
C04334=1068.166,242.079,412.887,173.664,30.113,155.468
C04335=1068.172,242.328,412.860,173.666,30.117,155.468
C04336=1068.178,242.576,412.833,173.668,30.121,155.469
C04337=1068.183,242.825,412.805,173.671,30.126,155.470
C04338=1068.190,243.073,412.778,173.673,30.129,155.470
C04339=1068.195,243.322,412.750,173.675,30.133,155.471
C04340=1068.202,243.570,412.723,173.678,30.138,155.472
C04341=1068.207,243.818,412.695,173.680,30.142,155.473
C04342=1068.213,244.067,412.668,173.682,30.145,155.473
C04343=1068.220,244.315,412.640,173.685,30.149,155.474
C04344=1068.225,244.564,412.613,173.687,30.154,155.475
C04345=1068.231,244.812,412.585,173.689,30.157,155.475
C04346=1068.237,245.060,412.557,173.691,30.161,155.476
C04347=1068.243,245.309,412.530,173.694,30.165,155.477
C04348=1068.248,245.557,412.502,173.697,30.170,155.477
C04349=1068.255,245.806,412.475,173.698,30.173,155.478
C04350=1068.260,246.054,412.447,173.701,30.177,155.479
C04351=1068.267,246.303,412.420,173.704,30.181,155.479
C04352=1068.272,246.551,412.392,173.705,30.185,155.480
C04353=1068.279,246.799,412.364,173.708,30.189,155.481
C04354=1068.284,247.047,412.336,173.710,30.193,155.481
C04355=1068.290,247.297,412.308,173.713,30.197,155.482
C04356=1068.296,247.545,412.281,173.715,30.201,155.483
C04357=1068.302,247.793,412.253,173.717,30.205,155.483
C04358=1068.307,248.041,412.225,173.720,30.210,155.484
C04359=1068.314,248.290,412.197,173.723,30.214,155.485
C04360=1068.319,248.538,412.169,173.724,30.217,155.486
C04361=1068.324,248.751,412.145,173.727,30.221,155.486
C04362=1068.329,248.963,412.122,173.729,30.224,155.487
C04363=1068.334,249.175,412.097,173.730,30.227,155.487
C04364=1068.339,249.388,412.074,173.733,30.231,155.488
C04365=1068.344,249.601,412.050,173.735,30.235,155.489
C04366=1068.349,249.812,412.026,173.736,30.238,155.489
C04367=1068.354,250.025,412.002,173.739,30.242,155.490
C04368=1068.358,250.237,411.978,173.741,30.245,155.490
C04369=1068.365,250.486,411.951,173.743,30.249,155.491
C04370=1068.370,250.734,411.923,173.746,30.253,155.492
C04371=1068.376,250.983,411.894,173.747,30.257,155.492
C04372=1068.382,251.231,411.867,173.750,30.261,155.493
C04373=1068.388,251.479,411.839,173.753,30.265,155.494
C04374=1068.394,251.728,411.810,173.755,30.269,155.494
C04375=1068.400,251.976,411.783,173.757,30.273,155.495
C04376=1068.406,252.224,411.753,173.760,30.277,155.496
C04377=1068.412,252.472,411.726,173.762,30.281,155.497
C04378=1068.418,252.721,411.698,173.765,30.285,155.497
C04379=1068.424,252.969,411.669,173.767,30.289,155.498
C04380=1068.429,253.217,411.641,173.769,30.293,155.499
C04381=1068.436,253.466,411.614,173.772,30.297,155.499
C04382=1068.442,253.715,411.585,173.774,30.301,155.500
C04383=1068.447,253.963,411.557,173.777,30.305,155.501
C04384=1068.453,254.211,411.529,173.779,30.309,155.501
C04385=1068.459,254.459,411.500,173.781,30.313,155.502
C04386=1068.465,254.707,411.473,173.784,30.317,155.503
C04387=1068.471,254.956,411.444,173.787,30.321,155.503
C04388=1068.477,255.205,411.416,173.789,30.325,155.504
C04389=1068.483,255.453,411.388,173.791,30.329,155.505
C04390=1068.489,255.701,411.359,173.793,30.333,155.505
C04391=1068.496,255.949,411.331,173.796,30.336,155.506
C04392=1068.501,256.197,411.303,173.799,30.341,155.507
C04393=1068.507,256.446,411.275,173.801,30.345,155.508
C04394=1068.513,256.694,411.246,173.803,30.348,155.508
C04395=1068.519,256.943,411.218,173.806,30.352,155.509
C04396=1068.525,257.191,411.190,173.808,30.356,155.509
C04397=1068.531,257.439,411.161,173.811,30.361,155.510
C04398=1068.537,257.688,411.133,173.814,30.365,155.511
C04399=1068.543,257.936,411.105,173.816,30.368,155.512
C04400=1068.549,258.184,411.076,173.818,30.372,155.512
C04401=1068.555,258.433,411.048,173.821,30.376,155.513
C04402=1068.561,258.681,411.019,173.823,30.380,155.514
C04403=1068.568,258.929,410.991,173.826,30.384,155.514
C04404=1068.574,259.178,410.963,173.828,30.388,155.515
C04405=1068.579,259.425,410.934,173.831,30.392,155.516
C04406=1068.585,259.674,410.906,173.833,30.396,155.516
C04407=1068.592,259.922,410.877,173.835,30.400,155.517
C04408=1068.597,260.171,410.848,173.838,30.404,155.518
C04409=1068.604,260.419,410.819,173.841,30.408,155.518
C04410=1068.610,260.668,410.791,173.843,30.412,155.519
C04411=1068.616,260.915,410.763,173.846,30.416,155.520
C04412=1068.622,261.164,410.734,173.849,30.419,155.520
C04413=1068.628,261.412,410.705,173.850,30.424,155.521
C04414=1068.634,261.661,410.677,173.853,30.428,155.522
C04415=1068.640,261.909,410.648,173.856,30.431,155.522
C04416=1068.646,262.157,410.620,173.858,30.435,155.523
C04417=1068.652,262.368,410.595,173.860,30.438,155.524
C04418=1068.657,262.579,410.572,173.863,30.442,155.524
C04419=1068.662,262.791,410.546,173.864,30.445,155.525
C04420=1068.667,263.002,410.523,173.867,30.449,155.525
C04421=1068.673,263.213,410.498,173.869,30.452,155.526
C04422=1068.678,263.424,410.473,173.872,30.455,155.526
C04423=1068.683,263.636,410.449,173.873,30.459,155.527
C04424=1068.688,263.847,410.424,173.876,30.462,155.528
C04425=1068.694,264.095,410.396,173.878,30.466,155.528
C04426=1068.700,264.343,410.367,173.880,30.470,155.529
C04427=1068.706,264.591,410.338,173.883,30.474,155.530
C04428=1068.712,264.839,410.309,173.886,30.478,155.530
C04429=1068.717,265.088,410.280,173.888,30.482,155.531
C04430=1068.724,265.336,410.251,173.891,30.486,155.532
C04431=1068.730,265.584,410.222,173.894,30.490,155.533
C04432=1068.736,265.833,410.193,173.896,30.495,155.533
C04433=1068.742,266.081,410.163,173.899,30.498,155.534
C04434=1068.748,266.330,410.135,173.901,30.502,155.535
C04435=1068.753,266.577,410.106,173.903,30.506,155.535
C04436=1068.759,266.825,410.077,173.906,30.510,155.536
C04437=1068.765,267.074,410.047,173.909,30.514,155.537
C04438=1068.771,267.322,410.018,173.911,30.518,155.537
C04439=1068.777,267.570,409.989,173.914,30.522,155.538
C04440=1068.784,267.818,409.960,173.916,30.526,155.539
C04441=1068.789,268.067,409.931,173.919,30.530,155.539
C04442=1068.795,268.315,409.902,173.922,30.535,155.540
C04443=1068.802,268.563,409.873,173.924,30.538,155.541
C04444=1068.808,268.811,409.844,173.927,30.542,155.542
C04445=1068.813,269.059,409.814,173.929,30.546,155.542
C04446=1068.820,269.308,409.785,173.931,30.550,155.543
C04447=1068.826,269.556,409.756,173.934,30.554,155.544
C04448=1068.831,269.804,409.726,173.937,30.558,155.544
C04449=1068.838,270.052,409.697,173.939,30.562,155.545
C04450=1068.844,270.300,409.668,173.942,30.566,155.546
C04451=1068.849,270.549,409.639,173.945,30.570,155.546
C04452=1068.856,270.797,409.609,173.947,30.575,155.547
C04453=1068.861,271.045,409.580,173.950,30.578,155.548
C04454=1068.867,271.294,409.551,173.953,30.582,155.549
C04455=1068.874,271.542,409.522,173.955,30.587,155.549
C04456=1068.879,271.790,409.492,173.958,30.590,155.550
C04457=1068.886,272.038,409.462,173.961,30.594,155.551
C04458=1068.891,272.286,409.433,173.963,30.599,155.551
C04459=1068.898,272.534,409.404,173.966,30.603,155.552
C04460=1068.903,272.783,409.374,173.968,30.606,155.553
C04461=1068.909,273.031,409.345,173.970,30.611,155.553
C04462=1068.915,273.279,409.315,173.973,30.614,155.554
C04463=1068.921,273.527,409.286,173.976,30.619,155.555
C04464=1068.927,273.775,409.256,173.978,30.623,155.556
C04465=1068.933,274.023,409.227,173.981,30.627,155.556
C04466=1068.939,274.271,409.197,173.984,30.631,155.557
C04467=1068.945,274.519,409.168,173.986,30.635,155.558
C04468=1068.951,274.768,409.138,173.989,30.639,155.558
C04469=1068.958,275.016,409.108,173.992,30.643,155.559
C04470=1068.963,275.264,409.078,173.994,30.647,155.560
C04471=1068.969,275.513,409.049,173.997,30.651,155.561
C04472=1068.975,275.760,409.019,174.000,30.655,155.561
C04473=1068.980,275.973,408.993,174.003,30.659,155.562
C04474=1068.986,276.186,408.968,174.004,30.662,155.562
C04475=1068.991,276.400,408.943,174.007,30.666,155.563
C04476=1068.996,276.612,408.916,174.009,30.669,155.564
C04477=1069.001,276.825,408.891,174.011,30.673,155.564
C04478=1069.006,277.038,408.866,174.013,30.676,155.565
C04479=1069.012,277.250,408.840,174.016,30.680,155.566
C04480=1069.017,277.464,408.814,174.019,30.683,155.566
C04481=1069.022,277.712,408.785,174.021,30.687,155.567
C04482=1069.029,277.960,408.755,174.024,30.691,155.568
C04483=1069.034,278.208,408.725,174.027,30.695,155.568
C04484=1069.040,278.456,408.695,174.029,30.699,155.569
C04485=1069.046,278.705,408.665,174.032,30.703,155.570
C04486=1069.053,278.953,408.635,174.035,30.708,155.570
C04487=1069.058,279.200,408.605,174.037,30.711,155.571
C04488=1069.064,279.449,408.575,174.040,30.715,155.572
C04489=1069.071,279.696,408.546,174.043,30.720,155.573
C04490=1069.077,279.945,408.516,174.045,30.723,155.573
C04491=1069.082,280.193,408.485,174.048,30.728,155.574
C04492=1069.089,280.441,408.455,174.051,30.732,155.575
C04493=1069.095,280.689,408.426,174.053,30.736,155.575
C04494=1069.100,280.937,408.395,174.056,30.740,155.576
C04495=1069.107,281.186,408.365,174.059,30.744,155.577
C04496=1069.113,281.433,408.334,174.061,30.748,155.577
C04497=1069.118,281.682,408.305,174.064,30.752,155.578
C04498=1069.124,281.930,408.274,174.067,30.756,155.579
C04499=1069.130,282.177,408.245,174.069,30.761,155.580
C04500=1069.137,282.426,408.214,174.072,30.764,155.580
C04501=1069.142,282.674,408.184,174.075,30.769,155.581
C04502=1069.148,282.922,408.154,174.078,30.773,155.582
C04503=1069.154,283.170,408.124,174.080,30.777,155.583
C04504=1069.160,283.418,408.093,174.083,30.781,155.583
C04505=1069.166,283.666,408.063,174.086,30.785,155.584
C04506=1069.172,283.914,408.032,174.088,30.789,155.585
C04507=1069.178,284.162,408.002,174.091,30.793,155.585
C04508=1069.184,284.411,407.972,174.094,30.797,155.586
C04509=1069.190,284.659,407.941,174.096,30.802,155.587
C04510=1069.196,284.907,407.911,174.099,30.806,155.588
C04511=1069.201,285.154,407.881,174.102,30.810,155.588
C04512=1069.209,285.403,407.851,174.104,30.814,155.589
C04513=1069.214,285.650,407.820,174.108,30.818,155.590
C04514=1069.220,285.898,407.790,174.111,30.822,155.591
C04515=1069.227,286.147,407.759,174.114,30.826,155.591
C04516=1069.233,286.395,407.729,174.116,30.831,155.592
C04517=1069.238,286.642,407.699,174.119,30.834,155.593
C04518=1069.245,286.891,407.668,174.122,30.839,155.593
C04519=1069.251,287.139,407.637,174.124,30.843,155.594
C04520=1069.257,287.387,407.607,174.127,30.847,155.595
C04521=1069.263,287.635,407.576,174.130,30.851,155.596
C04522=1069.269,287.882,407.545,174.132,30.855,155.596
C04523=1069.275,288.131,407.515,174.135,30.859,155.597
C04524=1069.281,288.379,407.484,174.139,30.864,155.598
C04525=1069.288,288.627,407.454,174.141,30.867,155.598
C04526=1069.293,288.875,407.423,174.144,30.872,155.599
C04527=1069.299,289.123,407.393,174.147,30.876,155.600
C04528=1069.306,289.371,407.362,174.150,30.880,155.601
C04529=1069.311,289.589,407.335,174.152,30.884,155.601
C04530=1069.316,289.807,407.308,174.154,30.887,155.602
C04531=1069.322,290.025,407.281,174.157,30.891,155.603
C04532=1069.327,290.243,407.254,174.159,30.894,155.603
C04533=1069.331,290.461,407.226,174.162,30.898,155.604
C04534=1069.337,290.680,407.199,174.164,30.902,155.605
C04535=1069.342,290.897,407.172,174.167,30.906,155.605
C04536=1069.347,291.115,407.145,174.169,30.909,155.606
C04537=1069.354,291.364,407.114,174.172,30.913,155.607
C04538=1069.360,291.611,407.083,174.175,30.918,155.607
C04539=1069.366,291.860,407.052,174.177,30.922,155.608
C04540=1069.371,292.108,407.021,174.180,30.926,155.609
C04541=1069.378,292.355,406.990,174.183,30.930,155.610
C04542=1069.384,292.603,406.960,174.187,30.935,155.610
C04543=1069.390,292.851,406.929,174.189,30.938,155.611
C04544=1069.396,293.099,406.897,174.192,30.943,155.612
C04545=1069.402,293.347,406.867,174.195,30.947,155.613
C04546=1069.408,293.595,406.835,174.197,30.951,155.613
C04547=1069.414,293.843,406.805,174.200,30.955,155.614
C04548=1069.420,294.091,406.773,174.203,30.959,155.615
C04549=1069.426,294.339,406.743,174.206,30.964,155.616
C04550=1069.433,294.587,406.711,174.209,30.968,155.616
C04551=1069.439,294.835,406.681,174.212,30.972,155.617
C04552=1069.445,295.083,406.649,174.215,30.976,155.618
C04553=1069.450,295.331,406.619,174.217,30.980,155.619
C04554=1069.457,295.579,406.587,174.220,30.985,155.619
C04555=1069.463,295.827,406.555,174.224,30.989,155.620
C04556=1069.469,296.075,406.525,174.226,30.993,155.621
C04557=1069.475,296.323,406.493,174.229,30.997,155.622
C04558=1069.481,296.570,406.462,174.232,31.002,155.622
C04559=1069.487,296.819,406.431,174.235,31.006,155.623
C04560=1069.493,297.066,406.399,174.238,31.010,155.624
C04561=1069.499,297.314,406.368,174.241,31.014,155.625
C04562=1069.505,297.562,406.337,174.244,31.019,155.625
C04563=1069.511,297.810,406.305,174.246,31.023,155.626
C04564=1069.517,298.058,406.274,174.249,31.027,155.627
C04565=1069.523,298.306,406.242,174.252,31.032,155.628
C04566=1069.529,298.553,406.211,174.256,31.036,155.629
C04567=1069.534,298.802,406.179,174.258,31.040,155.629
C04568=1069.540,299.050,406.147,174.261,31.045,155.630
C04569=1069.547,299.297,406.116,174.264,31.049,155.631
C04570=1069.553,299.546,406.084,174.266,31.053,155.632
C04571=1069.558,299.793,406.053,174.270,31.058,155.632
C04572=1069.565,300.041,406.021,174.273,31.062,155.633
C04573=1069.570,300.288,405.990,174.275,31.066,155.634
C04574=1069.576,300.537,405.957,174.278,31.071,155.635
C04575=1069.582,300.785,405.927,174.281,31.075,155.636
C04576=1069.588,301.033,405.895,174.285,31.079,155.636
C04577=1069.594,301.281,405.863,174.287,31.083,155.637
C04578=1069.600,301.528,405.832,174.290,31.088,155.638
C04579=1069.606,301.776,405.800,174.293,31.092,155.639
C04580=1069.612,302.025,405.768,174.296,31.096,155.639
C04581=1069.617,302.272,405.736,174.299,31.101,155.640
C04582=1069.624,302.520,405.705,174.302,31.105,155.641
C04583=1069.630,302.768,405.672,174.305,31.109,155.642
C04584=1069.636,303.015,405.640,174.307,31.114,155.643
C04585=1069.642,303.241,405.611,174.310,31.118,155.643
C04586=1069.647,303.466,405.583,174.313,31.122,155.644
C04587=1069.652,303.692,405.554,174.316,31.126,155.645
C04588=1069.658,303.918,405.525,174.318,31.130,155.646
C04589=1069.663,304.143,405.496,174.321,31.134,155.646
C04590=1069.669,304.369,405.467,174.324,31.137,155.647
C04591=1069.675,304.594,405.438,174.327,31.142,155.648
C04592=1069.680,304.820,405.409,174.329,31.146,155.648
C04593=1069.685,305.067,405.377,174.332,31.150,155.649
C04594=1069.692,305.315,405.345,174.336,31.154,155.650
C04595=1069.698,305.563,405.313,174.338,31.159,155.651
C04596=1069.704,305.811,405.281,174.341,31.163,155.651
C04597=1069.710,306.058,405.249,174.344,31.167,155.652
C04598=1069.717,306.306,405.217,174.348,31.172,155.653
C04599=1069.723,306.554,405.185,174.350,31.176,155.654
C04600=1069.729,306.802,405.153,174.353,31.180,155.655
C04601=1069.735,307.050,405.120,174.357,31.185,155.655
C04602=1069.740,307.297,405.089,174.360,31.189,155.656
C04603=1069.747,307.545,405.057,174.362,31.193,155.657
C04604=1069.753,307.793,405.024,174.366,31.198,155.658
C04605=1069.759,308.041,404.992,174.369,31.202,155.659
C04606=1069.766,308.289,404.960,174.371,31.207,155.659
C04607=1069.772,308.537,404.928,174.374,31.211,155.660
C04608=1069.778,308.785,404.896,174.378,31.215,155.661
C04609=1069.784,309.032,404.864,174.381,31.220,155.662
C04610=1069.790,309.280,404.832,174.383,31.224,155.663
C04611=1069.796,309.527,404.799,174.387,31.229,155.663
C04612=1069.802,309.776,404.767,174.390,31.233,155.664
C04613=1069.809,310.023,404.734,174.393,31.238,155.665
C04614=1069.815,310.271,404.703,174.396,31.242,155.666
C04615=1069.822,310.519,404.670,174.399,31.246,155.667
C04616=1069.828,310.767,404.638,174.402,31.251,155.667
C04617=1069.834,311.014,404.605,174.405,31.255,155.668
C04618=1069.840,311.262,404.573,174.408,31.259,155.669
C04619=1069.846,311.510,404.541,174.411,31.264,155.670
C04620=1069.853,311.758,404.508,174.415,31.268,155.671
C04621=1069.859,312.006,404.476,174.417,31.272,155.671
C04622=1069.866,312.253,404.444,174.420,31.277,155.672
C04623=1069.872,312.501,404.411,174.424,31.281,155.673
C04624=1069.878,312.749,404.379,174.427,31.286,155.674
C04625=1069.884,312.997,404.346,174.429,31.290,155.675
C04626=1069.890,313.244,404.313,174.433,31.295,155.675
C04627=1069.896,313.493,404.281,174.436,31.299,155.676
C04628=1069.903,313.740,404.249,174.440,31.303,155.677
C04629=1069.909,313.988,404.216,174.442,31.308,155.678
C04630=1069.915,314.235,404.183,174.445,31.312,155.679
C04631=1069.921,314.484,404.151,174.449,31.317,155.679
C04632=1069.928,314.731,404.118,174.452,31.321,155.680
C04633=1069.933,314.979,404.085,174.454,31.326,155.681
C04634=1069.939,315.227,404.052,174.458,31.331,155.682
C04635=1069.946,315.474,404.019,174.461,31.335,155.683
C04636=1069.951,315.722,403.986,174.464,31.340,155.684
C04637=1069.958,315.970,403.953,174.467,31.344,155.684
C04638=1069.963,316.218,403.920,174.470,31.349,155.685
C04639=1069.969,316.465,403.887,174.474,31.353,155.686
C04640=1069.976,316.713,403.855,174.476,31.358,155.687
C04641=1069.981,316.941,403.825,174.479,31.362,155.688
C04642=1069.986,317.168,403.794,174.482,31.367,155.689
C04643=1069.992,317.394,403.764,174.485,31.370,155.689
C04644=1069.998,317.622,403.733,174.488,31.375,155.690
C04645=1070.003,317.849,403.703,174.490,31.379,155.691
C04646=1070.009,318.077,403.673,174.493,31.383,155.692
C04647=1070.014,318.304,403.643,174.497,31.388,155.693
C04648=1070.019,318.531,403.612,174.500,31.392,155.693
C04649=1070.026,318.779,403.579,174.502,31.396,155.694
C04650=1070.031,319.026,403.546,174.506,31.401,155.695
C04651=1070.038,319.274,403.512,174.509,31.406,155.696
C04652=1070.045,319.522,403.480,174.512,31.410,155.697
C04653=1070.050,319.770,403.446,174.515,31.415,155.698
C04654=1070.056,320.017,403.413,174.518,31.420,155.698
C04655=1070.062,320.265,403.380,174.522,31.425,155.699
C04656=1070.068,320.513,403.347,174.525,31.429,155.700
C04657=1070.074,320.760,403.313,174.527,31.434,155.701
C04658=1070.081,321.008,403.280,174.531,31.438,155.702
C04659=1070.087,321.256,403.247,174.534,31.443,155.703
C04660=1070.093,321.504,403.214,174.538,31.448,155.704
C04661=1070.099,321.751,403.180,174.540,31.452,155.705
C04662=1070.105,321.999,403.147,174.544,31.457,155.705
C04663=1070.111,322.247,403.114,174.547,31.461,155.706
C04664=1070.118,322.494,403.080,174.550,31.466,155.707
C04665=1070.123,322.742,403.047,174.553,31.471,155.708
C04666=1070.130,322.989,403.013,174.556,31.475,155.709
C04667=1070.136,323.238,402.980,174.560,31.480,155.710
C04668=1070.142,323.485,402.947,174.563,31.485,155.711
C04669=1070.148,323.733,402.913,174.566,31.490,155.711
C04670=1070.155,323.980,402.880,174.569,31.494,155.712
C04671=1070.161,324.228,402.846,174.573,31.499,155.713
C04672=1070.167,324.476,402.813,174.576,31.504,155.714
C04673=1070.173,324.723,402.779,174.579,31.509,155.715
C04674=1070.180,324.971,402.746,174.582,31.513,155.716
C04675=1070.186,325.219,402.712,174.586,31.518,155.717
C04676=1070.192,325.466,402.679,174.589,31.523,155.718
C04677=1070.199,325.714,402.645,174.592,31.527,155.719
C04678=1070.205,325.962,402.612,174.595,31.532,155.719
C04679=1070.211,326.209,402.578,174.599,31.537,155.720
C04680=1070.217,326.457,402.543,174.602,31.541,155.721
C04681=1070.224,326.705,402.511,174.605,31.546,155.722
C04682=1070.230,326.953,402.476,174.608,31.551,155.723
C04683=1070.236,327.200,402.443,174.612,31.556,155.724
C04684=1070.242,327.448,402.409,174.615,31.560,155.725
C04685=1070.249,327.695,402.376,174.619,31.565,155.726
C04686=1070.255,327.942,402.342,174.621,31.570,155.726
C04687=1070.261,328.191,402.308,174.625,31.575,155.727
C04688=1070.268,328.438,402.274,174.628,31.579,155.728
C04689=1070.275,328.686,402.240,174.632,31.584,155.729
C04690=1070.281,328.933,402.207,174.634,31.589,155.730
C04691=1070.287,329.182,402.173,174.638,31.593,155.731
C04692=1070.293,329.429,402.139,174.641,31.598,155.732
C04693=1070.300,329.677,402.105,174.645,31.603,155.733
C04694=1070.306,329.924,402.071,174.647,31.608,155.734
C04695=1070.313,330.172,402.036,174.651,31.613,155.735
C04696=1070.319,330.419,402.003,174.655,31.618,155.736
C04697=1070.325,330.644,401.972,174.658,31.622,155.736
C04698=1070.331,330.868,401.941,174.661,31.626,155.737
C04699=1070.336,331.092,401.911,174.663,31.631,155.738
C04700=1070.342,331.316,401.881,174.667,31.635,155.739
C04701=1070.348,331.541,401.849,174.670,31.640,155.740
C04702=1070.353,331.764,401.817,174.673,31.644,155.740
C04703=1070.359,331.988,401.787,174.676,31.648,155.741
C04704=1070.364,332.212,401.756,174.678,31.653,155.742
C04705=1070.371,332.460,401.722,174.682,31.658,155.743
C04706=1070.376,332.708,401.688,174.686,31.663,155.744
C04707=1070.383,332.956,401.653,174.689,31.668,155.745
C04708=1070.389,333.202,401.618,174.692,31.672,155.746
C04709=1070.396,333.450,401.585,174.695,31.677,155.747
C04710=1070.402,333.697,401.551,174.699,31.682,155.748
C04711=1070.409,333.945,401.516,174.702,31.687,155.749
C04712=1070.415,334.193,401.482,174.706,31.692,155.750
C04713=1070.421,334.440,401.448,174.709,31.697,155.751
C04714=1070.428,334.688,401.413,174.712,31.702,155.752
C04715=1070.434,334.935,401.378,174.716,31.707,155.752
C04716=1070.440,335.183,401.344,174.719,31.712,155.753
C04717=1070.445,335.431,401.309,174.722,31.717,155.754
C04718=1070.452,335.678,401.274,174.726,31.722,155.755
C04719=1070.458,335.926,401.240,174.729,31.727,155.756
C04720=1070.464,336.173,401.206,174.733,31.732,155.757
C04721=1070.471,336.421,401.171,174.737,31.737,155.758
C04722=1070.477,336.669,401.136,174.739,31.742,155.759
C04723=1070.483,336.916,401.102,174.743,31.747,155.760
C04724=1070.490,337.163,401.067,174.746,31.752,155.761
C04725=1070.497,337.411,401.033,174.750,31.757,155.762
C04726=1070.502,337.659,400.999,174.754,31.763,155.763
C04727=1070.509,337.906,400.963,174.756,31.767,155.764
C04728=1070.516,338.154,400.929,174.760,31.772,155.765
C04729=1070.521,338.401,400.894,174.764,31.778,155.766
C04730=1070.528,338.649,400.859,174.767,31.782,155.767
C04731=1070.534,338.896,400.824,174.771,31.788,155.768
C04732=1070.540,339.144,400.790,174.774,31.793,155.769
C04733=1070.546,339.391,400.754,174.777,31.798,155.770
C04734=1070.553,339.639,400.719,174.781,31.803,155.771
C04735=1070.559,339.887,400.685,174.785,31.808,155.772
C04736=1070.566,340.133,400.650,174.787,31.814,155.773
C04737=1070.572,340.381,400.614,174.791,31.819,155.774
C04738=1070.578,340.629,400.580,174.795,31.824,155.775
C04739=1070.584,340.876,400.545,174.798,31.829,155.776
C04740=1070.590,341.123,400.509,174.802,31.834,155.777
C04741=1070.597,341.371,400.475,174.805,31.839,155.778
C04742=1070.604,341.619,400.440,174.808,31.844,155.779
C04743=1070.610,341.866,400.405,174.812,31.850,155.780
C04744=1070.616,342.113,400.369,174.816,31.855,155.781
C04745=1070.622,342.361,400.335,174.820,31.860,155.782
C04746=1070.629,342.608,400.300,174.822,31.865,155.783
C04747=1070.635,342.856,400.264,174.826,31.870,155.784
C04748=1070.642,343.103,400.229,174.830,31.876,155.785
C04749=1070.649,343.351,400.194,174.833,31.881,155.786
C04750=1070.654,343.598,400.159,174.837,31.886,155.787
C04751=1070.660,343.846,400.124,174.840,31.891,155.788
C04752=1070.667,344.093,400.089,174.844,31.897,155.789
C04753=1070.673,344.315,400.056,174.847,31.901,155.790
C04754=1070.678,344.537,400.025,174.850,31.906,155.791
C04755=1070.684,344.758,399.994,174.854,31.911,155.792
C04756=1070.690,344.979,399.961,174.857,31.916,155.793
C04757=1070.695,345.201,399.930,174.859,31.920,155.794
C04758=1070.701,345.423,399.899,174.863,31.925,155.795
C04759=1070.706,345.644,399.866,174.866,31.930,155.795
C04760=1070.712,345.866,399.835,174.869,31.935,155.796
C04761=1070.719,346.114,399.800,174.873,31.940,155.797
C04762=1070.725,346.361,399.764,174.877,31.945,155.798
C04763=1070.731,346.609,399.729,174.880,31.950,155.799
C04764=1070.738,346.856,399.692,174.883,31.956,155.800
C04765=1070.745,347.103,399.657,174.887,31.961,155.802
C04766=1070.751,347.351,399.621,174.891,31.966,155.803
C04767=1070.757,347.598,399.586,174.895,31.972,155.804
C04768=1070.763,347.846,399.550,174.897,31.978,155.805
C04769=1070.770,348.093,399.514,174.901,31.983,155.806
C04770=1070.776,348.340,399.479,174.905,31.988,155.807
C04771=1070.782,348.587,399.444,174.909,31.994,155.808
C04772=1070.788,348.834,399.407,174.913,31.999,155.809
C04773=1070.795,349.081,399.372,174.916,32.004,155.810
C04774=1070.801,349.329,399.336,174.919,32.010,155.811
C04775=1070.807,349.576,399.300,174.923,32.015,155.812
C04776=1070.814,349.824,399.265,174.927,32.021,155.813
C04777=1070.821,350.072,399.229,174.931,32.027,155.814
C04778=1070.827,350.319,399.192,174.935,32.032,155.815
C04779=1070.834,350.566,399.157,174.938,32.037,155.816
C04780=1070.840,350.813,399.121,174.941,32.043,155.818
C04781=1070.846,351.061,399.085,174.945,32.049,155.819
C04782=1070.853,351.308,399.049,174.949,32.054,155.820
C04783=1070.859,351.556,399.013,174.953,32.059,155.821
C04784=1070.866,351.803,398.977,174.957,32.065,155.822
C04785=1070.872,352.050,398.941,174.960,32.070,155.823
C04786=1070.879,352.297,398.905,174.963,32.076,155.824
C04787=1070.885,352.545,398.869,174.967,32.082,155.825
C04788=1070.891,352.792,398.833,174.971,32.087,155.826
C04789=1070.898,353.039,398.797,174.975,32.093,155.828
C04790=1070.904,353.287,398.760,174.979,32.098,155.829
C04791=1070.910,353.534,398.724,174.982,32.104,155.830
C04792=1070.917,353.781,398.688,174.985,32.110,155.831
C04793=1070.923,354.029,398.652,174.989,32.115,155.832
C04794=1070.930,354.276,398.616,174.993,32.121,155.833
C04795=1070.936,354.523,398.580,174.997,32.127,155.834
C04796=1070.943,354.770,398.543,175.001,32.132,155.835
C04797=1070.949,355.017,398.507,175.005,32.138,155.836
C04798=1070.956,355.265,398.471,175.008,32.144,155.838
C04799=1070.962,355.512,398.434,175.011,32.149,155.839
C04800=1070.968,355.759,398.398,175.015,32.155,155.840
C04801=1070.975,356.006,398.361,175.019,32.161,155.841
C04802=1070.981,356.253,398.325,175.023,32.166,155.842
C04803=1070.988,356.501,398.288,175.027,32.172,155.843
C04804=1070.994,356.748,398.252,175.030,32.178,155.844
C04805=1071.001,356.995,398.215,175.034,32.183,155.846
C04806=1071.007,357.242,398.179,175.038,32.189,155.847
C04807=1071.014,357.490,398.142,175.042,32.195,155.848
C04808=1071.020,357.737,398.105,175.046,32.201,155.849
C04809=1071.026,357.961,398.072,175.049,32.206,155.850
C04810=1071.031,358.184,398.040,175.053,32.212,155.851
C04811=1071.038,358.407,398.006,175.056,32.216,155.852
C04812=1071.044,358.631,397.973,175.059,32.222,155.853
C04813=1071.050,358.855,397.940,175.062,32.227,155.854
C04814=1071.056,359.077,397.907,175.066,32.232,155.855
C04815=1071.062,359.301,397.874,175.070,32.238,155.856
C04816=1071.067,359.525,397.841,175.073,32.243,155.857
C04817=1071.074,359.772,397.804,175.077,32.249,155.859
C04818=1071.080,360.019,397.767,175.081,32.255,155.860
C04819=1071.087,360.267,397.730,175.084,32.260,155.861
C04820=1071.093,360.514,397.693,175.088,32.266,155.862
C04821=1071.100,360.760,397.656,175.092,32.272,155.863
C04822=1071.107,361.008,397.619,175.096,32.279,155.865
C04823=1071.113,361.255,397.583,175.100,32.284,155.866
C04824=1071.120,361.501,397.546,175.104,32.290,155.867
C04825=1071.126,361.749,397.508,175.108,32.296,155.868
C04826=1071.132,361.997,397.472,175.112,32.302,155.869
C04827=1071.139,362.244,397.434,175.115,32.308,155.871
C04828=1071.146,362.491,397.398,175.119,32.314,155.872
C04829=1071.152,362.737,397.360,175.123,32.320,155.873
C04830=1071.158,362.985,397.323,175.127,32.326,155.874
C04831=1071.165,363.232,397.286,175.131,32.332,155.875
C04832=1071.172,363.479,397.249,175.135,32.338,155.877
C04833=1071.178,363.726,397.212,175.139,32.344,155.878
C04834=1071.185,363.974,397.175,175.143,32.350,155.879
C04835=1071.192,364.220,397.138,175.147,32.356,155.880
C04836=1071.199,364.467,397.100,175.150,32.362,155.882
C04837=1071.204,364.715,397.063,175.154,32.369,155.883
C04838=1071.212,364.962,397.025,175.158,32.374,155.884
C04839=1071.218,365.209,396.988,175.162,32.381,155.885
C04840=1071.224,365.456,396.951,175.166,32.387,155.887
C04841=1071.230,365.703,396.913,175.170,32.393,155.888
C04842=1071.237,365.950,396.876,175.174,32.399,155.889
C04843=1071.244,366.197,396.838,175.178,32.405,155.890
C04844=1071.250,366.444,396.801,175.182,32.412,155.892
C04845=1071.256,366.692,396.763,175.185,32.418,155.893
C04846=1071.263,366.938,396.726,175.190,32.424,155.894
C04847=1071.270,367.185,396.688,175.194,32.430,155.895
C04848=1071.277,367.433,396.651,175.198,32.437,155.897
C04849=1071.283,367.679,396.613,175.202,32.443,155.898
C04850=1071.290,367.926,396.575,175.206,32.449,155.899
C04851=1071.296,368.173,396.537,175.210,32.455,155.901
C04852=1071.303,368.420,396.500,175.214,32.462,155.902
C04853=1071.309,368.667,396.462,175.218,32.468,155.903
C04854=1071.316,368.914,396.425,175.222,32.474,155.905
C04855=1071.323,369.162,396.387,175.225,32.481,155.906
C04856=1071.329,369.408,396.349,175.229,32.487,155.907
C04857=1071.336,369.656,396.311,175.234,32.493,155.908
C04858=1071.342,369.902,396.274,175.238,32.499,155.910
C04859=1071.349,370.149,396.236,175.242,32.506,155.911
C04860=1071.356,370.397,396.198,175.246,32.512,155.912
C04861=1071.362,370.643,396.161,175.250,32.518,155.914
C04862=1071.369,370.891,396.123,175.254,32.525,155.915
C04863=1071.376,371.137,396.084,175.258,32.532,155.916
C04864=1071.383,371.385,396.046,175.262,32.538,155.918
C04865=1071.388,371.616,396.011,175.266,32.544,155.919
C04866=1071.395,371.848,395.975,175.270,32.550,155.920
C04867=1071.402,372.080,395.940,175.274,32.556,155.921
C04868=1071.408,372.312,395.904,175.277,32.562,155.923
C04869=1071.414,372.544,395.868,175.281,32.568,155.924
C04870=1071.420,372.776,395.832,175.285,32.574,155.925
C04871=1071.426,373.008,395.796,175.289,32.580,155.926
C04872=1071.433,373.240,395.760,175.293,32.587,155.928
C04873=1071.440,373.487,395.723,175.297,32.593,155.929
C04874=1071.447,373.734,395.684,175.301,32.600,155.931
C04875=1071.453,373.980,395.646,175.305,32.606,155.932
C04876=1071.459,374.227,395.607,175.309,32.613,155.933
C04877=1071.466,374.475,395.569,175.314,32.619,155.935
C04878=1071.473,374.721,395.530,175.318,32.626,155.936
C04879=1071.479,374.968,395.493,175.322,32.633,155.937
C04880=1071.485,375.215,395.454,175.326,32.640,155.939
C04881=1071.493,375.462,395.415,175.330,32.646,155.940
C04882=1071.499,375.709,395.377,175.335,32.653,155.942
C04883=1071.506,375.956,395.338,175.339,32.660,155.943
C04884=1071.513,376.203,395.300,175.343,32.667,155.944
C04885=1071.519,376.449,395.262,175.347,32.673,155.946
C04886=1071.526,376.696,395.223,175.351,32.680,155.947
C04887=1071.533,376.943,395.184,175.355,32.687,155.949
C04888=1071.539,377.190,395.145,175.359,32.693,155.950
C04889=1071.546,377.437,395.107,175.363,32.700,155.952
C04890=1071.553,377.684,395.068,175.368,32.707,155.953
C04891=1071.560,377.931,395.030,175.372,32.714,155.954
C04892=1071.566,378.178,394.991,175.376,32.720,155.956
C04893=1071.573,378.425,394.952,175.380,32.727,155.957
C04894=1071.580,378.671,394.913,175.385,32.734,155.959
C04895=1071.587,378.918,394.874,175.389,32.741,155.960
C04896=1071.594,379.165,394.835,175.393,32.748,155.962
C04897=1071.600,379.411,394.797,175.397,32.755,155.963
C04898=1071.607,379.658,394.758,175.402,32.762,155.964
C04899=1071.613,379.905,394.719,175.406,32.769,155.966
C04900=1071.621,380.152,394.680,175.410,32.776,155.967
C04901=1071.628,380.399,394.641,175.415,32.783,155.969
C04902=1071.634,380.646,394.602,175.419,32.790,155.970
C04903=1071.641,380.893,394.564,175.423,32.796,155.972
C04904=1071.648,381.140,394.525,175.428,32.803,155.973
C04905=1071.655,381.386,394.485,175.432,32.811,155.975
C04906=1071.662,381.633,394.446,175.436,32.818,155.976
C04907=1071.669,381.880,394.407,175.441,32.825,155.978
C04908=1071.676,382.126,394.369,175.445,32.832,155.979
C04909=1071.682,382.373,394.328,175.449,32.839,155.981
C04910=1071.689,382.620,394.290,175.454,32.846,155.982
C04911=1071.696,382.867,394.251,175.458,32.853,155.984
C04912=1071.702,383.113,394.211,175.462,32.860,155.985
C04913=1071.709,383.360,394.172,175.467,32.868,155.987
C04914=1071.716,383.606,394.132,175.471,32.875,155.988
C04915=1071.723,383.853,394.093,175.475,32.882,155.990
C04916=1071.729,384.101,394.054,175.480,32.889,155.991
C04917=1071.737,384.347,394.014,175.484,32.897,155.993
C04918=1071.743,384.594,393.975,175.489,32.904,155.995
C04919=1071.750,384.840,393.935,175.493,32.911,155.996
C04920=1071.757,385.086,393.896,175.497,32.919,155.998
C04921=1071.762,385.313,393.860,175.501,32.925,155.999
C04922=1071.769,385.540,393.823,175.505,32.932,156.001
C04923=1071.775,385.766,393.786,175.510,32.939,156.002
C04924=1071.782,385.994,393.751,175.514,32.945,156.004
C04925=1071.788,386.220,393.714,175.518,32.952,156.005
C04926=1071.795,386.447,393.678,175.522,32.959,156.006
C04927=1071.801,386.674,393.641,175.526,32.966,156.008
C04928=1071.807,386.901,393.605,175.530,32.972,156.009
C04929=1071.814,387.147,393.565,175.535,32.980,156.011
C04930=1071.822,387.394,393.525,175.540,32.987,156.013
C04931=1071.828,387.640,393.485,175.544,32.994,156.014
C04932=1071.835,387.887,393.445,175.549,33.002,156.016
C04933=1071.842,388.135,393.406,175.553,33.010,156.017
C04934=1071.849,388.381,393.366,175.558,33.017,156.019
C04935=1071.856,388.627,393.327,175.562,33.024,156.021
C04936=1071.863,388.874,393.286,175.567,33.032,156.022
C04937=1071.870,389.120,393.246,175.571,33.040,156.024
C04938=1071.877,389.367,393.206,175.576,33.048,156.026
C04939=1071.884,389.614,393.166,175.580,33.055,156.027
C04940=1071.891,389.860,393.126,175.585,33.062,156.029
C04941=1071.899,390.147,393.080,175.590,33.071,156.031
C04942=1071.907,390.433,393.033,175.595,33.080,156.033
C04943=1071.916,390.720,392.987,175.600,33.089,156.035
C04944=1071.924,391.005,392.940,175.607,33.098,156.036
C04945=1071.931,391.252,392.900,175.611,33.105,156.038
C04946=1071.938,391.499,392.860,175.616,33.113,156.040
C04947=1071.945,391.746,392.819,175.620,33.121,156.042
C04948=1071.952,391.991,392.779,175.625,33.129,156.043
C04949=1071.959,392.239,392.739,175.629,33.137,156.045
C04950=1071.965,392.485,392.698,175.634,33.145,156.047
C04951=1071.973,392.731,392.658,175.639,33.153,156.048
C04952=1071.980,392.978,392.618,175.643,33.160,156.050
C04953=1071.987,393.225,392.577,175.648,33.168,156.052
C04954=1071.994,393.471,392.536,175.653,33.176,156.054
C04955=1072.001,393.718,392.496,175.658,33.184,156.055
C04956=1072.008,393.964,392.455,175.662,33.192,156.057
C04957=1072.015,394.211,392.415,175.667,33.200,156.059
C04958=1072.022,394.457,392.374,175.672,33.208,156.060
C04959=1072.029,394.704,392.334,175.676,33.216,156.062
C04960=1072.036,394.950,392.293,175.681,33.224,156.064
C04961=1072.043,395.197,392.253,175.685,33.232,156.066
C04962=1072.050,395.444,392.212,175.691,33.240,156.067
C04963=1072.057,395.689,392.171,175.696,33.248,156.069
C04964=1072.064,395.937,392.130,175.700,33.256,156.071
C04965=1072.071,396.183,392.089,175.705,33.264,156.073
C04966=1072.078,396.429,392.048,175.710,33.272,156.075
C04967=1072.086,396.675,392.007,175.714,33.281,156.076
C04968=1072.093,396.923,391.967,175.719,33.289,156.078
C04969=1072.100,397.169,391.926,175.724,33.297,156.080
C04970=1072.107,397.415,391.885,175.729,33.305,156.082
C04971=1072.114,397.662,391.844,175.734,33.314,156.084
C04972=1072.122,397.908,391.802,175.739,33.322,156.086
C04973=1072.128,398.154,391.762,175.743,33.330,156.087
C04974=1072.135,398.401,391.720,175.748,33.339,156.089
C04975=1072.143,398.647,391.679,175.754,33.347,156.091
C04976=1072.150,398.894,391.638,175.758,33.355,156.093
C04977=1072.157,399.156,391.594,175.763,33.364,156.095
C04978=1072.164,399.418,391.550,175.768,33.373,156.097
C04979=1072.172,399.681,391.507,175.773,33.382,156.099
C04980=1072.180,399.943,391.463,175.779,33.391,156.101
C04981=1072.187,400.189,391.421,175.784,33.400,156.103
C04982=1072.194,400.435,391.380,175.789,33.408,156.105
C04983=1072.201,400.682,391.338,175.794,33.416,156.107
C04984=1072.208,400.929,391.297,175.798,33.425,156.109
C04985=1072.216,401.175,391.256,175.804,33.433,156.110
C04986=1072.223,401.421,391.214,175.809,33.442,156.112
C04987=1072.231,401.668,391.173,175.814,33.451,156.114
C04988=1072.237,401.915,391.131,175.818,33.459,156.116
C04989=1072.245,402.161,391.089,175.823,33.468,156.118
C04990=1072.252,402.407,391.048,175.829,33.477,156.120
C04991=1072.259,402.654,391.006,175.834,33.485,156.122
C04992=1072.267,402.900,390.965,175.839,33.494,156.124
C04993=1072.273,403.147,390.923,175.843,33.502,156.126
C04994=1072.281,403.393,390.881,175.849,33.511,156.128
C04995=1072.288,403.639,390.840,175.854,33.520,156.130
C04996=1072.295,403.886,390.797,175.859,33.529,156.132
C04997=1072.303,404.132,390.755,175.864,33.538,156.134
C04998=1072.310,404.378,390.714,175.870,33.547,156.136
C04999=1072.317,404.624,390.671,175.874,33.556,156.138
C05000=1072.324,404.871,390.630,175.879,33.565,156.140
C05001=1072.332,405.117,390.588,175.884,33.574,156.142
C05002=1072.339,405.363,390.546,175.890,33.582,156.144
C05003=1072.346,405.609,390.504,175.895,33.592,156.146
C05004=1072.353,405.857,390.461,175.900,33.601,156.148
C05005=1072.361,406.103,390.419,175.906,33.610,156.150
C05006=1072.368,406.349,390.377,175.911,33.619,156.152
C05007=1072.375,406.595,390.335,175.916,33.628,156.154
C05008=1072.382,406.841,390.292,175.921,33.637,156.156
C05009=1072.390,407.087,390.251,175.927,33.646,156.158
C05010=1072.397,407.334,390.208,175.931,33.655,156.160
C05011=1072.405,407.580,390.166,175.936,33.665,156.162
C05012=1072.412,407.827,390.123,175.942,33.674,156.164
C05013=1072.419,408.073,390.081,175.947,33.683,156.167
C05014=1072.426,408.319,390.039,175.952,33.692,156.169
C05015=1072.434,408.566,389.996,175.958,33.702,156.171
C05016=1072.441,408.812,389.954,175.963,33.711,156.173
C05017=1072.448,409.058,389.911,175.968,33.721,156.175
C05018=1072.455,409.304,389.868,175.974,33.730,156.177
C05019=1072.463,409.550,389.826,175.979,33.739,156.179
C05020=1072.470,409.797,389.783,175.984,33.749,156.182
C05021=1072.477,410.043,389.741,175.990,33.758,156.184
C05022=1072.486,410.289,389.698,175.995,33.768,156.186
C05023=1072.493,410.535,389.655,176.002,33.777,156.188
C05024=1072.499,410.782,389.612,176.007,33.787,156.190
C05025=1072.508,411.028,389.569,176.012,33.796,156.192
C05026=1072.515,411.274,389.527,176.018,33.806,156.195
C05027=1072.523,411.520,389.483,176.023,33.815,156.197
C05028=1072.529,411.767,389.441,176.028,33.825,156.199
C05029=1072.538,412.013,389.398,176.034,33.835,156.201
C05030=1072.545,412.259,389.355,176.039,33.844,156.203
C05031=1072.552,412.505,389.312,176.045,33.854,156.206
C05032=1072.560,412.751,389.269,176.050,33.864,156.208
C05033=1072.568,413.017,389.222,176.057,33.874,156.210
C05034=1072.577,413.282,389.176,176.063,33.885,156.213
C05035=1072.584,413.548,389.129,176.068,33.895,156.215
C05036=1072.593,413.813,389.083,176.075,33.906,156.218
C05037=1072.601,414.060,389.040,176.080,33.916,156.220
C05038=1072.608,414.307,388.997,176.086,33.926,156.222
C05039=1072.615,414.552,388.953,176.091,33.935,156.224
C05040=1072.623,414.799,388.910,176.098,33.946,156.227
C05041=1072.631,415.044,388.867,176.103,33.956,156.229
C05042=1072.639,415.291,388.824,176.109,33.966,156.231
C05043=1072.646,415.537,388.780,176.114,33.976,156.234
C05044=1072.654,415.783,388.737,176.121,33.986,156.236
C05045=1072.661,416.029,388.693,176.126,33.996,156.239
C05046=1072.668,416.276,388.649,176.132,34.006,156.241
C05047=1072.676,416.521,388.606,176.137,34.016,156.243
C05048=1072.683,416.768,388.562,176.144,34.026,156.246
C05049=1072.691,417.013,388.518,176.149,34.037,156.248
C05050=1072.699,417.259,388.474,176.155,34.047,156.250
C05051=1072.706,417.505,388.431,176.161,34.057,156.253
C05052=1072.714,417.752,388.387,176.167,34.068,156.255
C05053=1072.722,417.997,388.343,176.172,34.078,156.258
C05054=1072.729,418.243,388.299,176.179,34.089,156.260
C05055=1072.737,418.489,388.255,176.184,34.099,156.262
C05056=1072.745,418.735,388.212,176.190,34.110,156.265
C05057=1072.753,418.982,388.168,176.196,34.120,156.267
C05058=1072.760,419.227,388.123,176.202,34.131,156.270
C05059=1072.767,419.473,388.080,176.209,34.141,156.272
C05060=1072.776,419.719,388.035,176.214,34.152,156.275
C05061=1072.784,419.965,387.991,176.221,34.162,156.277
C05062=1072.791,420.211,387.947,176.226,34.173,156.280
C05063=1072.799,420.457,387.903,176.232,34.183,156.282
C05064=1072.807,420.703,387.859,176.239,34.194,156.285
C05065=1072.814,420.949,387.815,176.244,34.205,156.287
C05066=1072.823,421.195,387.770,176.251,34.216,156.290
C05067=1072.831,421.441,387.726,176.256,34.226,156.292
C05068=1072.838,421.688,387.682,176.263,34.237,156.295
C05069=1072.846,421.933,387.637,176.269,34.248,156.298
C05070=1072.854,422.179,387.593,176.275,34.259,156.300
C05071=1072.861,422.425,387.548,176.281,34.270,156.303
C05072=1072.869,422.670,387.504,176.288,34.281,156.305
C05073=1072.876,422.916,387.459,176.293,34.292,156.308
C05074=1072.885,423.163,387.414,176.300,34.303,156.311
C05075=1072.893,423.408,387.370,176.307,34.314,156.313
C05076=1072.900,423.654,387.324,176.312,34.326,156.316
C05077=1072.908,423.900,387.280,176.319,34.337,156.319
C05078=1072.916,424.146,387.235,176.325,34.348,156.321
C05079=1072.924,424.391,387.191,176.332,34.359,156.324
C05080=1072.931,424.637,387.146,176.338,34.371,156.327
C05081=1072.939,424.883,387.101,176.344,34.382,156.329
C05082=1072.947,425.129,387.056,176.351,34.393,156.332
C05083=1072.955,425.374,387.012,176.357,34.404,156.335
C05084=1072.964,425.620,386.966,176.363,34.415,156.337
C05085=1072.971,425.866,386.921,176.370,34.427,156.340
C05086=1072.980,426.111,386.876,176.377,34.438,156.343
C05087=1072.987,426.357,386.831,176.383,34.450,156.346
C05088=1072.996,426.603,386.786,176.389,34.461,156.348
C05089=1073.005,426.887,386.734,176.397,34.475,156.351
C05090=1073.014,427.171,386.682,176.404,34.488,156.355
C05091=1073.023,427.455,386.629,176.412,34.502,156.358
C05092=1073.032,427.739,386.577,176.420,34.515,156.361
C05093=1073.041,427.985,386.531,176.426,34.527,156.364
C05094=1073.048,428.231,386.486,176.433,34.538,156.367
C05095=1073.056,428.476,386.441,176.440,34.551,156.370
C05096=1073.065,428.723,386.395,176.446,34.562,156.373
C05097=1073.072,428.968,386.349,176.453,34.574,156.375
C05098=1073.080,429.213,386.304,176.459,34.586,156.378
C05099=1073.089,429.459,386.258,176.466,34.598,156.381
C05100=1073.096,429.705,386.212,176.473,34.610,156.384
C05101=1073.105,429.951,386.166,176.480,34.622,156.387
C05102=1073.112,430.196,386.121,176.487,34.634,156.390
C05103=1073.121,430.441,386.076,176.494,34.646,156.393
C05104=1073.129,430.687,386.029,176.501,34.658,156.396
C05105=1073.137,430.932,385.983,176.508,34.670,156.399
C05106=1073.145,431.179,385.937,176.514,34.682,156.402
C05107=1073.153,431.425,385.891,176.521,34.695,156.405
C05108=1073.162,431.669,385.846,176.527,34.707,156.408
C05109=1073.170,431.915,385.800,176.534,34.719,156.411
C05110=1073.178,432.161,385.754,176.541,34.732,156.414
C05111=1073.186,432.406,385.707,176.548,34.744,156.417
C05112=1073.194,432.652,385.662,176.555,34.757,156.420
C05113=1073.203,432.897,385.615,176.562,34.769,156.423
C05114=1073.211,433.142,385.568,176.570,34.782,156.426
C05115=1073.219,433.388,385.522,176.577,34.795,156.429
C05116=1073.227,433.634,385.475,176.584,34.807,156.432
C05117=1073.235,433.879,385.429,176.592,34.820,156.435
C05118=1073.243,434.125,385.383,176.599,34.833,156.438
C05119=1073.251,434.370,385.336,176.606,34.845,156.441
C05120=1073.259,434.615,385.290,176.613,34.858,156.445
C05121=1073.268,434.861,385.243,176.620,34.871,156.448
C05122=1073.276,435.106,385.196,176.627,34.884,156.451
C05123=1073.285,435.352,385.149,176.634,34.897,156.454
C05124=1073.294,435.597,385.103,176.641,34.910,156.457
C05125=1073.301,435.842,385.056,176.650,34.922,156.460
C05126=1073.310,436.088,385.010,176.657,34.936,156.464
C05127=1073.319,436.333,384.963,176.664,34.949,156.467
C05128=1073.326,436.579,384.916,176.671,34.962,156.470
C05129=1073.335,436.824,384.869,176.678,34.975,156.473
C05130=1073.344,437.069,384.821,176.686,34.988,156.477
C05131=1073.352,437.315,384.775,176.694,35.001,156.480
C05132=1073.361,437.560,384.728,176.701,35.015,156.483
C05133=1073.369,437.806,384.681,176.708,35.028,156.487
C05134=1073.378,438.050,384.634,176.716,35.041,156.490
C05135=1073.386,438.297,384.586,176.724,35.055,156.493
C05136=1073.395,438.541,384.539,176.731,35.068,156.497
C05137=1073.403,438.787,384.492,176.739,35.081,156.500
C05138=1073.412,439.032,384.445,176.746,35.095,156.503
C05139=1073.420,439.278,384.398,176.754,35.109,156.507
C05140=1073.429,439.523,384.350,176.762,35.123,156.510
C05141=1073.438,439.767,384.303,176.769,35.136,156.514
C05142=1073.446,440.013,384.255,176.778,35.150,156.517
C05143=1073.454,440.258,384.208,176.785,35.164,156.520
C05144=1073.463,440.503,384.160,176.793,35.178,156.524
C05145=1073.476,440.872,384.089,176.805,35.199,156.529
C05146=1073.489,441.239,384.017,176.817,35.219,156.534
C05147=1073.501,441.608,383.945,176.829,35.241,156.540
C05148=1073.515,441.975,383.873,176.840,35.262,156.545
C05149=1073.524,442.220,383.825,176.849,35.276,156.549
C05150=1073.532,442.466,383.777,176.856,35.290,156.552
C05151=1073.540,442.711,383.729,176.865,35.304,156.556
C05152=1073.550,442.955,383.681,176.873,35.319,156.560
C05153=1073.558,443.201,383.632,176.881,35.333,156.563
C05154=1073.567,443.446,383.585,176.889,35.347,156.567
C05155=1073.576,443.691,383.536,176.897,35.362,156.570
C05156=1073.585,443.936,383.488,176.905,35.376,156.574
C05157=1073.593,444.181,383.439,176.914,35.391,156.578
C05158=1073.602,444.427,383.391,176.922,35.406,156.582
C05159=1073.611,444.671,383.343,176.930,35.420,156.585
C05160=1073.620,444.917,383.294,176.939,35.435,156.589
C05161=1073.628,445.162,383.246,176.948,35.450,156.593
C05162=1073.637,445.406,383.197,176.955,35.464,156.597
C05163=1073.647,445.651,383.148,176.964,35.479,156.600
C05164=1073.656,445.896,383.099,176.973,35.494,156.604
C05165=1073.664,446.141,383.051,176.981,35.509,156.608
C05166=1073.673,446.387,383.002,176.989,35.525,156.612
C05167=1073.682,446.631,382.954,176.998,35.540,156.616
C05168=1073.691,446.876,382.905,177.006,35.554,156.620
C05169=1073.700,447.121,382.855,177.015,35.570,156.624
C05170=1073.709,447.366,382.806,177.024,35.585,156.627
C05171=1073.718,447.611,382.757,177.032,35.600,156.631
C05172=1073.727,447.856,382.709,177.040,35.615,156.635
C05173=1073.736,448.100,382.659,177.048,35.630,156.639
C05174=1073.745,448.344,382.611,177.054,35.646,156.643
C05175=1073.754,448.588,382.562,177.061,35.660,156.647
C05176=1073.765,448.833,382.514,177.068,35.675,156.651
C05177=1073.776,449.078,382.466,177.075,35.690,156.654
C05178=1073.790,449.322,382.419,177.081,35.703,156.658
C05179=1073.803,449.568,382.373,177.087,35.716,156.661
C05180=1073.819,449.814,382.328,177.094,35.728,156.665
C05181=1073.465,449.811,382.085,177.076,35.877,156.704
C05182=1073.450,449.565,382.130,177.070,35.864,156.701
C05183=1073.435,449.320,382.176,177.064,35.851,156.697
C05184=1073.422,449.076,382.223,177.057,35.838,156.694
C05185=1073.410,448.831,382.271,177.050,35.824,156.690
C05186=1073.399,448.586,382.319,177.043,35.809,156.686
C05187=1073.390,448.341,382.368,177.036,35.794,156.683
C05188=1073.381,448.097,382.417,177.028,35.779,156.679
C05189=1073.371,447.853,382.465,177.022,35.764,156.675
C05190=1073.363,447.609,382.515,177.013,35.749,156.671
C05191=1073.354,447.364,382.564,177.005,35.734,156.667
C05192=1073.345,447.119,382.613,176.996,35.719,156.663
C05193=1073.336,446.874,382.662,176.987,35.703,156.659
C05194=1073.326,446.629,382.710,176.979,35.688,156.655
C05195=1073.317,446.384,382.760,176.970,35.673,156.651
C05196=1073.308,446.139,382.809,176.961,35.658,156.647
C05197=1073.300,445.894,382.857,176.953,35.643,156.643
C05198=1073.291,445.649,382.907,176.944,35.628,156.640
C05199=1073.282,445.405,382.955,176.936,35.613,156.636
C05200=1073.273,445.159,383.004,176.927,35.599,156.632
C05201=1073.264,444.915,383.053,176.919,35.584,156.628
C05202=1073.255,444.669,383.100,176.910,35.569,156.624
C05203=1073.247,444.425,383.149,176.902,35.555,156.621
C05204=1073.237,444.179,383.198,176.893,35.540,156.617
C05205=1073.229,443.934,383.246,176.885,35.526,156.613
C05206=1073.220,443.689,383.295,176.877,35.511,156.610
C05207=1073.211,443.444,383.343,176.868,35.496,156.606
C05208=1073.202,443.200,383.391,176.860,35.482,156.602
C05209=1073.194,442.954,383.439,176.852,35.468,156.599
C05210=1073.184,442.709,383.488,176.844,35.453,156.595
C05211=1073.176,442.464,383.536,176.836,35.439,156.591
C05212=1073.167,442.219,383.583,176.827,35.425,156.588
C05213=1073.159,441.973,383.632,176.819,35.411,156.584
C05214=1073.146,441.624,383.701,176.808,35.391,156.579
C05215=1073.134,441.274,383.769,176.796,35.370,156.574
C05216=1073.121,440.924,383.837,176.785,35.351,156.569
C05217=1073.109,440.574,383.905,176.773,35.331,156.564
C05218=1073.100,440.329,383.953,176.766,35.317,156.560
C05219=1073.092,440.083,384.001,176.757,35.303,156.557
C05220=1073.083,439.838,384.048,176.750,35.289,156.554
C05221=1073.075,439.593,384.096,176.742,35.276,156.550
C05222=1073.066,439.348,384.143,176.734,35.262,156.547
C05223=1073.057,439.103,384.191,176.727,35.248,156.543
C05224=1073.049,438.857,384.238,176.719,35.235,156.540
C05225=1073.041,438.612,384.286,176.711,35.222,156.537
C05226=1073.032,438.367,384.332,176.703,35.208,156.533
C05227=1073.023,438.122,384.380,176.696,35.195,156.530
C05228=1073.014,437.876,384.427,176.688,35.182,156.527
C05229=1073.007,437.631,384.474,176.680,35.168,156.523
C05230=1072.997,437.385,384.522,176.673,35.155,156.520
C05231=1072.989,437.140,384.569,176.665,35.141,156.516
C05232=1072.981,436.895,384.615,176.658,35.128,156.513
C05233=1072.972,436.650,384.662,176.650,35.115,156.510
C05234=1072.964,436.404,384.709,176.643,35.102,156.507
C05235=1072.955,436.159,384.756,176.635,35.089,156.503
C05236=1072.947,435.913,384.804,176.628,35.076,156.500
C05237=1072.938,435.668,384.850,176.620,35.063,156.497
C05238=1072.930,435.422,384.897,176.613,35.050,156.494
C05239=1072.921,435.177,384.944,176.606,35.037,156.491
C05240=1072.913,434.932,384.990,176.599,35.024,156.487
C05241=1072.905,434.687,385.037,176.591,35.012,156.484
C05242=1072.896,434.441,385.084,176.583,34.999,156.481
C05243=1072.888,434.195,385.130,176.576,34.986,156.478
C05244=1072.880,433.951,385.177,176.569,34.973,156.475
C05245=1072.871,433.705,385.223,176.562,34.961,156.472
C05246=1072.863,433.459,385.269,176.555,34.948,156.469
C05247=1072.855,433.214,385.316,176.548,34.935,156.466
C05248=1072.847,432.968,385.362,176.540,34.923,156.462
C05249=1072.838,432.723,385.409,176.533,34.910,156.459
C05250=1072.831,432.477,385.455,176.526,34.898,156.456
C05251=1072.823,432.231,385.501,176.519,34.885,156.453
C05252=1072.815,431.986,385.548,176.512,34.873,156.450
C05253=1072.807,431.740,385.594,176.505,34.861,156.447
C05254=1072.797,431.495,385.640,176.498,34.848,156.444
C05255=1072.790,431.250,385.686,176.491,34.836,156.441
C05256=1072.781,431.004,385.732,176.484,34.824,156.438
C05257=1072.773,430.759,385.778,176.477,34.812,156.435
C05258=1072.765,430.513,385.824,176.470,34.800,156.432
C05259=1072.757,430.268,385.869,176.463,34.788,156.429
C05260=1072.749,430.021,385.915,176.457,34.775,156.426
C05261=1072.741,429.776,385.961,176.450,34.763,156.423
C05262=1072.732,429.530,386.007,176.443,34.752,156.421
C05263=1072.724,429.285,386.053,176.436,34.739,156.418
C05264=1072.716,429.039,386.099,176.429,34.727,156.415
C05265=1072.708,428.794,386.144,176.422,34.716,156.412
C05266=1072.701,428.548,386.190,176.416,34.704,156.409
C05267=1072.692,428.302,386.235,176.409,34.692,156.406
C05268=1072.684,428.056,386.280,176.402,34.680,156.403
C05269=1072.677,427.811,386.326,176.395,34.668,156.401
C05270=1072.667,427.525,386.380,176.387,34.655,156.397
C05271=1072.657,427.240,386.432,176.380,34.641,156.394
C05272=1072.648,426.954,386.484,176.372,34.628,156.391
C05273=1072.638,426.668,386.536,176.364,34.615,156.388
C05274=1072.631,426.422,386.582,176.359,34.603,156.385
C05275=1072.622,426.177,386.627,176.352,34.591,156.382
C05276=1072.614,425.930,386.672,176.345,34.580,156.379
C05277=1072.606,425.685,386.718,176.339,34.569,156.377
C05278=1072.599,425.439,386.762,176.332,34.557,156.374
C05279=1072.590,425.194,386.808,176.325,34.546,156.371
C05280=1072.583,424.948,386.852,176.320,34.535,156.368
C05281=1072.574,424.701,386.897,176.313,34.524,156.366
C05282=1072.567,424.456,386.943,176.306,34.512,156.363
C05283=1072.559,424.210,386.987,176.300,34.501,156.360
C05284=1072.551,423.964,387.032,176.293,34.490,156.358
C05285=1072.543,423.719,387.076,176.287,34.479,156.355
C05286=1072.535,423.473,387.121,176.281,34.468,156.352
C05287=1072.527,423.227,387.166,176.274,34.456,156.350
C05288=1072.519,422.982,387.211,176.268,34.446,156.347
C05289=1072.512,422.736,387.256,176.262,34.434,156.344
C05290=1072.504,422.490,387.300,176.256,34.423,156.342
C05291=1072.497,422.244,387.345,176.249,34.412,156.339
C05292=1072.489,421.998,387.389,176.244,34.402,156.337
C05293=1072.481,421.752,387.434,176.237,34.390,156.334
C05294=1072.473,421.506,387.479,176.231,34.380,156.331
C05295=1072.465,421.260,387.523,176.224,34.369,156.329
C05296=1072.457,421.014,387.566,176.219,34.358,156.326
C05297=1072.449,420.768,387.611,176.212,34.347,156.324
C05298=1072.442,420.522,387.656,176.206,34.337,156.321
C05299=1072.434,420.277,387.700,176.200,34.326,156.319
C05300=1072.426,420.030,387.744,176.194,34.315,156.316
C05301=1072.418,419.784,387.788,176.187,34.305,156.314
C05302=1072.410,419.539,387.832,176.182,34.294,156.311
C05303=1072.402,419.292,387.876,176.176,34.284,156.309
C05304=1072.395,419.046,387.921,176.169,34.273,156.306
C05305=1072.387,418.800,387.965,176.164,34.263,156.304
C05306=1072.380,418.555,388.009,176.157,34.252,156.301
C05307=1072.372,418.309,388.052,176.152,34.242,156.299
C05308=1072.364,418.063,388.096,176.146,34.231,156.296
C05309=1072.356,417.816,388.140,176.139,34.221,156.294
C05310=1072.348,417.570,388.184,176.134,34.211,156.292
C05311=1072.341,417.325,388.228,176.128,34.201,156.289
C05312=1072.333,417.079,388.271,176.122,34.190,156.287
C05313=1072.325,416.832,388.315,176.116,34.180,156.284
C05314=1072.318,416.586,388.359,176.111,34.170,156.282
C05315=1072.311,416.341,388.403,176.105,34.159,156.280
C05316=1072.303,416.094,388.447,176.098,34.149,156.277
C05317=1072.295,415.848,388.490,176.093,34.139,156.275
C05318=1072.288,415.602,388.534,176.087,34.129,156.273
C05319=1072.280,415.356,388.577,176.081,34.119,156.270
C05320=1072.273,415.110,388.620,176.075,34.109,156.268
C05321=1072.265,414.864,388.664,176.070,34.099,156.266
C05322=1072.257,414.618,388.707,176.064,34.089,156.263
C05323=1072.250,414.372,388.750,176.059,34.079,156.261
C05324=1072.242,414.126,388.794,176.052,34.069,156.259
C05325=1072.234,413.879,388.838,176.047,34.059,156.256
C05326=1072.226,413.612,388.884,176.041,34.048,156.254
C05327=1072.218,413.345,388.930,176.035,34.038,156.251
C05328=1072.209,413.078,388.978,176.028,34.027,156.249
C05329=1072.201,412.810,389.024,176.023,34.017,156.247
C05330=1072.193,412.564,389.068,176.017,34.007,156.244
C05331=1072.186,412.318,389.110,176.011,33.997,156.242
C05332=1072.178,412.072,389.153,176.005,33.987,156.240
C05333=1072.171,411.826,389.197,176.000,33.978,156.238
C05334=1072.163,411.579,389.240,175.994,33.968,156.235
C05335=1072.156,411.333,389.283,175.989,33.959,156.233
C05336=1072.148,411.087,389.325,175.983,33.949,156.231
C05337=1072.141,410.841,389.368,175.978,33.940,156.229
C05338=1072.134,410.595,389.411,175.972,33.930,156.227
C05339=1072.126,410.348,389.453,175.967,33.920,156.224
C05340=1072.119,410.102,389.497,175.962,33.911,156.222
C05341=1072.111,409.855,389.539,175.956,33.902,156.220
C05342=1072.104,409.610,389.581,175.951,33.892,156.218
C05343=1072.096,409.364,389.625,175.945,33.883,156.216
C05344=1072.089,409.117,389.668,175.940,33.874,156.214
C05345=1072.081,408.871,389.709,175.935,33.864,156.211
C05346=1072.075,408.625,389.752,175.929,33.855,156.209
C05347=1072.067,408.379,389.795,175.924,33.846,156.207
C05348=1072.059,408.132,389.838,175.918,33.836,156.205
C05349=1072.052,407.886,389.880,175.913,33.827,156.203
C05350=1072.045,407.640,389.922,175.908,33.818,156.201
C05351=1072.038,407.394,389.965,175.902,33.808,156.199
C05352=1072.030,407.147,390.008,175.897,33.799,156.197
C05353=1072.023,406.901,390.049,175.892,33.790,156.194
C05354=1072.016,406.654,390.092,175.886,33.781,156.192
C05355=1072.008,406.409,390.134,175.881,33.772,156.190
C05356=1072.002,406.162,390.176,175.876,33.763,156.188
C05357=1071.993,405.916,390.219,175.870,33.754,156.186
C05358=1071.987,405.669,390.261,175.865,33.745,156.184
C05359=1071.979,405.423,390.303,175.859,33.735,156.182
C05360=1071.972,405.176,390.345,175.855,33.727,156.180
C05361=1071.965,404.930,390.387,175.850,33.718,156.178
C05362=1071.957,404.684,390.429,175.845,33.709,156.176
C05363=1071.951,404.438,390.471,175.839,33.700,156.174
C05364=1071.943,404.192,390.513,175.834,33.691,156.172
C05365=1071.936,403.945,390.554,175.829,33.682,156.170
C05366=1071.928,403.698,390.597,175.823,33.673,156.168
C05367=1071.921,403.452,390.639,175.819,33.664,156.166
C05368=1071.913,403.205,390.680,175.814,33.656,156.164
C05369=1071.906,402.959,390.723,175.808,33.647,156.162
C05370=1071.899,402.713,390.764,175.803,33.638,156.160
C05371=1071.892,402.467,390.806,175.798,33.630,156.158
C05372=1071.884,402.220,390.847,175.794,33.621,156.156
C05373=1071.877,401.974,390.889,175.788,33.613,156.154
C05374=1071.870,401.727,390.931,175.783,33.604,156.152
C05375=1071.863,401.480,390.972,175.778,33.595,156.150
C05376=1071.855,401.234,391.014,175.772,33.587,156.149
C05377=1071.848,400.988,391.055,175.768,33.578,156.147
C05378=1071.841,400.742,391.096,175.763,33.569,156.145
C05379=1071.834,400.495,391.137,175.758,33.561,156.143
C05380=1071.826,400.249,391.179,175.752,33.552,156.141
C05381=1071.820,400.003,391.221,175.748,33.544,156.139
C05382=1071.812,399.738,391.265,175.743,33.535,156.137
C05383=1071.804,399.475,391.309,175.738,33.526,156.135
C05384=1071.796,399.211,391.353,175.732,33.517,156.133
C05385=1071.789,398.948,391.398,175.727,33.508,156.131
C05386=1071.782,398.701,391.439,175.722,33.500,156.129
C05387=1071.775,398.454,391.481,175.717,33.491,156.127
C05388=1071.768,398.208,391.521,175.712,33.483,156.125
C05389=1071.760,397.962,391.562,175.707,33.475,156.124
C05390=1071.753,397.716,391.603,175.702,33.466,156.122
C05391=1071.746,397.469,391.645,175.698,33.458,156.120
C05392=1071.739,397.222,391.685,175.693,33.450,156.118
C05393=1071.732,396.976,391.726,175.687,33.442,156.116
C05394=1071.725,396.729,391.767,175.683,33.434,156.114
C05395=1071.717,396.483,391.808,175.678,33.425,156.113
C05396=1071.711,396.237,391.849,175.673,33.417,156.111
C05397=1071.703,395.990,391.890,175.669,33.409,156.109
C05398=1071.696,395.743,391.931,175.663,33.401,156.107
C05399=1071.690,395.497,391.972,175.658,33.393,156.106
C05400=1071.682,395.251,392.012,175.654,33.385,156.104
C05401=1071.675,395.004,392.053,175.649,33.377,156.102
C05402=1071.668,394.758,392.094,175.645,33.369,156.100
C05403=1071.661,394.511,392.135,175.640,33.361,156.098
C05404=1071.654,394.265,392.175,175.634,33.353,156.097
C05405=1071.647,394.018,392.216,175.630,33.345,156.095
C05406=1071.639,393.771,392.256,175.625,33.337,156.093
C05407=1071.633,393.525,392.297,175.621,33.329,156.091
C05408=1071.626,393.278,392.338,175.616,33.321,156.090
C05409=1071.619,393.032,392.379,175.612,33.313,156.088
C05410=1071.611,392.785,392.419,175.606,33.305,156.086
C05411=1071.605,392.539,392.459,175.601,33.297,156.084
C05412=1071.598,392.292,392.500,175.597,33.289,156.083
C05413=1071.591,392.046,392.539,175.592,33.282,156.081
C05414=1071.584,391.799,392.580,175.588,33.274,156.079
C05415=1071.577,391.553,392.621,175.583,33.266,156.078
C05416=1071.569,391.306,392.661,175.579,33.259,156.076
C05417=1071.563,391.059,392.701,175.573,33.251,156.074
C05418=1071.556,390.812,392.741,175.569,33.243,156.073
C05419=1071.548,390.567,392.782,175.564,33.236,156.071
C05420=1071.541,390.319,392.822,175.560,33.228,156.069
C05421=1071.534,390.073,392.862,175.555,33.220,156.068
C05422=1071.527,389.827,392.901,175.551,33.213,156.066
C05423=1071.520,389.580,392.942,175.546,33.205,156.064
C05424=1071.513,389.334,392.981,175.542,33.197,156.063
C05425=1071.506,389.086,393.022,175.537,33.190,156.061
C05426=1071.499,388.840,393.061,175.532,33.182,156.059
C05427=1071.493,388.594,393.102,175.527,33.175,156.058
C05428=1071.485,388.347,393.141,175.523,33.168,156.056
C05429=1071.478,388.100,393.181,175.518,33.160,156.055
C05430=1071.471,387.854,393.221,175.514,33.152,156.053
C05431=1071.464,387.607,393.261,175.509,33.145,156.051
C05432=1071.457,387.361,393.301,175.505,33.138,156.050
C05433=1071.450,387.114,393.340,175.500,33.130,156.048
C05434=1071.443,386.867,393.380,175.496,33.123,156.047
C05435=1071.436,386.620,393.420,175.492,33.115,156.045
C05436=1071.429,386.374,393.460,175.486,33.108,156.043
C05437=1071.423,386.127,393.499,175.482,33.100,156.042
C05438=1071.415,385.879,393.539,175.477,33.093,156.040
C05439=1071.408,385.631,393.579,175.473,33.086,156.039
C05440=1071.402,385.383,393.618,175.468,33.078,156.037
C05441=1071.395,385.134,393.658,175.464,33.071,156.035
C05442=1071.388,384.888,393.699,175.460,33.064,156.034
C05443=1071.381,384.641,393.737,175.455,33.056,156.032
C05444=1071.374,384.395,393.777,175.451,33.049,156.031
C05445=1071.367,384.149,393.817,175.446,33.042,156.029
C05446=1071.360,383.901,393.856,175.442,33.035,156.028
C05447=1071.353,383.655,393.896,175.438,33.027,156.026
C05448=1071.347,383.408,393.935,175.433,33.020,156.025
C05449=1071.340,383.161,393.974,175.429,33.013,156.023
C05450=1071.333,382.915,394.014,175.425,33.006,156.021
C05451=1071.327,382.668,394.053,175.420,32.999,156.020
C05452=1071.320,382.421,394.093,175.415,32.992,156.018
C05453=1071.313,382.174,394.132,175.411,32.985,156.017
C05454=1071.307,381.928,394.170,175.406,32.977,156.015
C05455=1071.300,381.681,394.211,175.402,32.971,156.014
C05456=1071.293,381.434,394.249,175.398,32.963,156.012
C05457=1071.287,381.187,394.288,175.393,32.956,156.011
